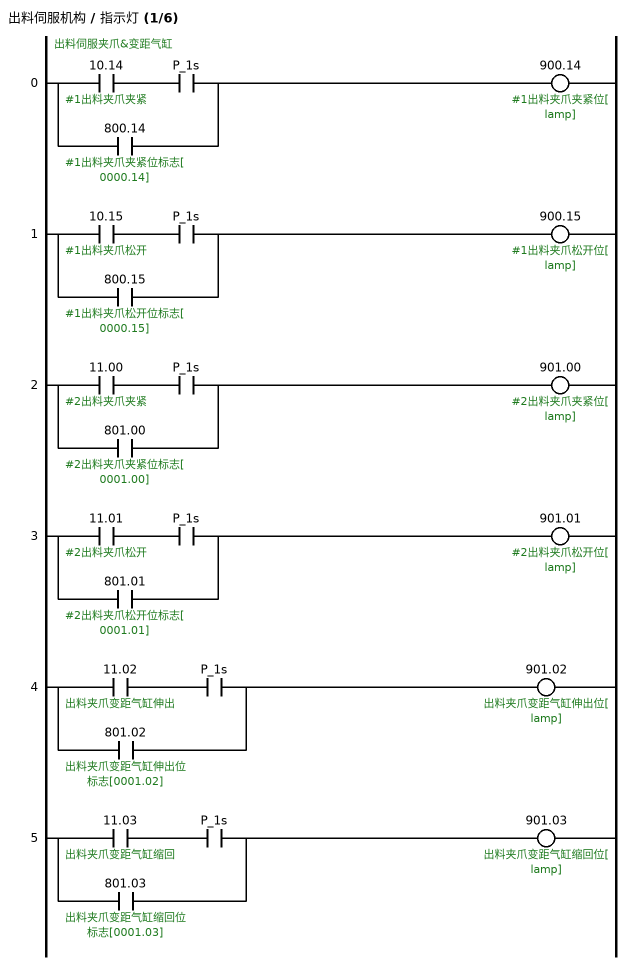
; [picture p504: 出料伺服机构 / 指示灯, rungs 0-5]
; rung 0: 出料伺服夹爪&变距气缸
LD 10.14  ; #1出料夹爪夹紧
AND P_1s
OR 800.14  ; #1出料夹爪夹紧位标志[0000.14]
OUT 900.14  ; #1出料夹爪夹紧位[lamp]
; rung 1
LD 10.15  ; #1出料夹爪松开
AND P_1s
OR 800.15  ; #1出料夹爪松开位标志[0000.15]
OUT 900.15  ; #1出料夹爪松开位[lamp]
; rung 2
LD 11.00  ; #2出料夹爪夹紧
AND P_1s
OR 801.00  ; #2出料夹爪夹紧位标志[0001.00]
OUT 901.00  ; #2出料夹爪夹紧位[lamp]
; rung 3
LD 11.01  ; #2出料夹爪松开
AND P_1s
OR 801.01  ; #2出料夹爪松开位标志[0001.01]
OUT 901.01  ; #2出料夹爪松开位[lamp]
; rung 4
LD 11.02  ; 出料夹爪变距气缸伸出
AND P_1s
OR 801.02  ; 出料夹爪变距气缸伸出位标志[0001.02]
OUT 901.02  ; 出料夹爪变距气缸伸出位[lamp]
; rung 5
LD 11.03  ; 出料夹爪变距气缸缩回
AND P_1s
OR 801.03  ; 出料夹爪变距气缸缩回位标志[0001.03]
OUT 901.03  ; 出料夹爪变距气缸缩回位[lamp]

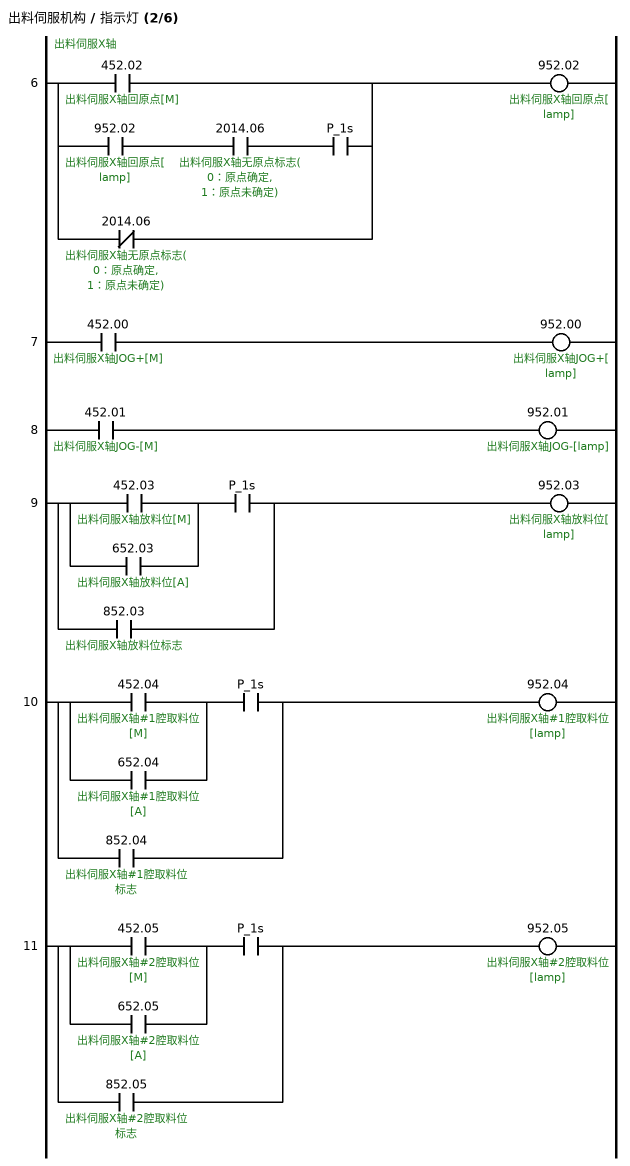
; rung 6: 出料伺服X轴
LD 452.02  ; 出料伺服X轴回原点[M]
LD 952.02  ; 出料伺服X轴回原点[lamp]
AND 2014.06  ; 出料伺服X轴无原点标志(0：原点确定,1：原点未确定)
AND P_1s
ORLD
ORNOT 2014.06  ; 出料伺服X轴无原点标志(0：原点确定,1：原点未确定)
OUT 952.02  ; 出料伺服X轴回原点[lamp]
; rung 7
LD 452.00  ; 出料伺服X轴JOG+[M]
OUT 952.00  ; 出料伺服X轴JOG+[lamp]
; rung 8
LD 452.01  ; 出料伺服X轴JOG-[M]
OUT 952.01  ; 出料伺服X轴JOG-[lamp]
; rung 9
LD 452.03  ; 出料伺服X轴放料位[M]
OR 652.03  ; 出料伺服X轴放料位[A]
AND P_1s
OR 852.03  ; 出料伺服X轴放料位标志
OUT 952.03  ; 出料伺服X轴放料位[lamp]
; rung 10
LD 452.04  ; 出料伺服X轴#1腔取料位[M]
OR 652.04  ; 出料伺服X轴#1腔取料位[A]
AND P_1s
OR 852.04  ; 出料伺服X轴#1腔取料位标志
OUT 952.04  ; 出料伺服X轴#1腔取料位[lamp]
; rung 11
LD 452.05  ; 出料伺服X轴#2腔取料位[M]
OR 652.05  ; 出料伺服X轴#2腔取料位[A]
AND P_1s
OR 852.05  ; 出料伺服X轴#2腔取料位标志
OUT 952.05  ; 出料伺服X轴#2腔取料位[lamp]

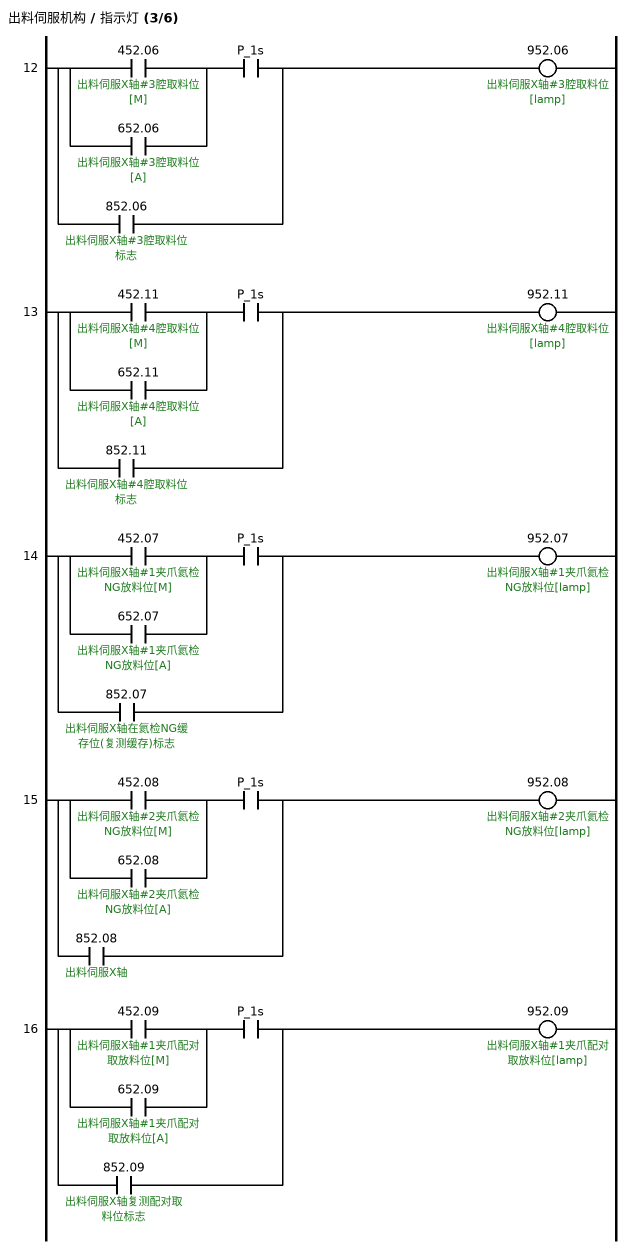
; rung 12
LD 452.06  ; 出料伺服X轴#3腔取料位[M]
OR 652.06  ; 出料伺服X轴#3腔取料位[A]
AND P_1s
OR 852.06  ; 出料伺服X轴#3腔取料位标志
OUT 952.06  ; 出料伺服X轴#3腔取料位[lamp]
; rung 13
LD 452.11  ; 出料伺服X轴#4腔取料位[M]
OR 652.11  ; 出料伺服X轴#4腔取料位[A]
AND P_1s
OR 852.11  ; 出料伺服X轴#4腔取料位标志
OUT 952.11  ; 出料伺服X轴#4腔取料位[lamp]
; rung 14
LD 452.07  ; 出料伺服X轴#1夹爪氦检NG放料位[M]
OR 652.07  ; 出料伺服X轴#1夹爪氦检NG放料位[A]
AND P_1s
OR 852.07  ; 出料伺服X轴在氦检NG缓存位(复测缓存)标志
OUT 952.07  ; 出料伺服X轴#1夹爪氦检NG放料位[lamp]
; rung 15
LD 452.08  ; 出料伺服X轴#2夹爪氦检NG放料位[M]
OR 652.08  ; 出料伺服X轴#2夹爪氦检NG放料位[A]
AND P_1s
OR 852.08  ; 出料伺服X轴
OUT 952.08  ; 出料伺服X轴#2夹爪氦检NG放料位[lamp]
; rung 16
LD 452.09  ; 出料伺服X轴#1夹爪配对取放料位[M]
OR 652.09  ; 出料伺服X轴#1夹爪配对取放料位[A]
AND P_1s
OR 852.09  ; 出料伺服X轴复测配对取料位标志
OUT 952.09  ; 出料伺服X轴#1夹爪配对取放料位[lamp]

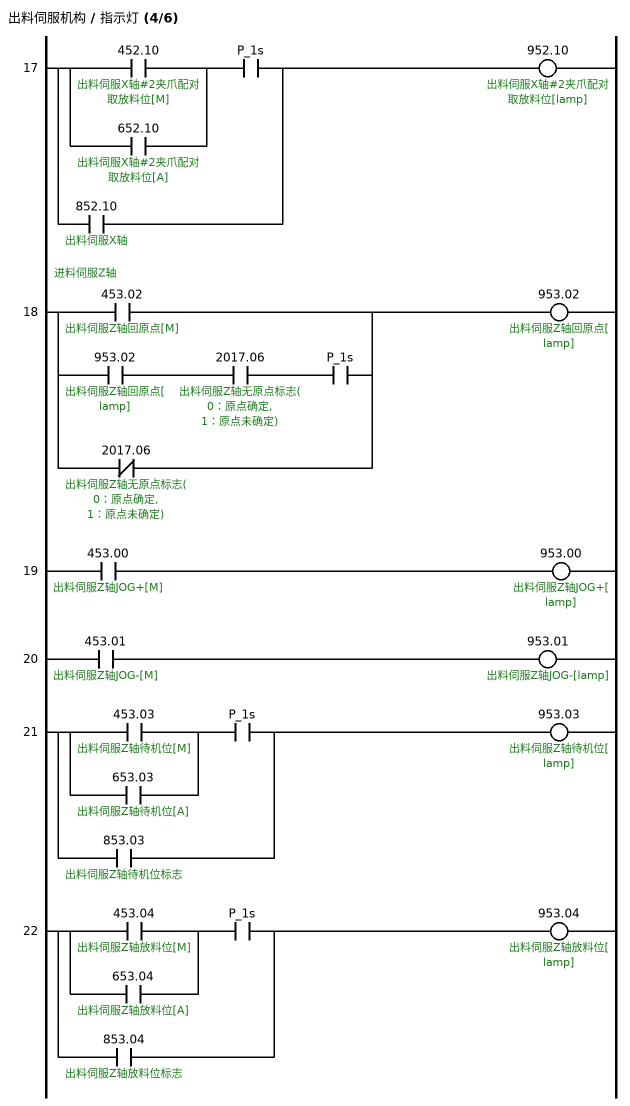
; rung 17
LD 452.10  ; 出料伺服X轴#2夹爪配对取放料位[M]
OR 652.10  ; 出料伺服X轴#2夹爪配对取放料位[A]
AND P_1s
OR 852.10  ; 出料伺服X轴
OUT 952.10  ; 出料伺服X轴#2夹爪配对取放料位[lamp]
; rung 18: 进料伺服Z轴
LD 453.02  ; 出料伺服Z轴回原点[M]
LD 953.02  ; 出料伺服Z轴回原点[lamp]
AND 2017.06  ; 出料伺服Z轴无原点标志(0：原点确定,1：原点未确定)
AND P_1s
ORLD
ORNOT 2017.06  ; 出料伺服Z轴无原点标志(0：原点确定,1：原点未确定)
OUT 953.02  ; 出料伺服Z轴回原点[lamp]
; rung 19
LD 453.00  ; 出料伺服Z轴JOG+[M]
OUT 953.00  ; 出料伺服Z轴JOG+[lamp]
; rung 20
LD 453.01  ; 出料伺服Z轴JOG-[M]
OUT 953.01  ; 出料伺服Z轴JOG-[lamp]
; rung 21
LD 453.03  ; 出料伺服Z轴待机位[M]
OR 653.03  ; 出料伺服Z轴待机位[A]
AND P_1s
OR 853.03  ; 出料伺服Z轴待机位标志
OUT 953.03  ; 出料伺服Z轴待机位[lamp]
; rung 22
LD 453.04  ; 出料伺服Z轴放料位[M]
OR 653.04  ; 出料伺服Z轴放料位[A]
AND P_1s
OR 853.04  ; 出料伺服Z轴放料位标志
OUT 953.04  ; 出料伺服Z轴放料位[lamp]

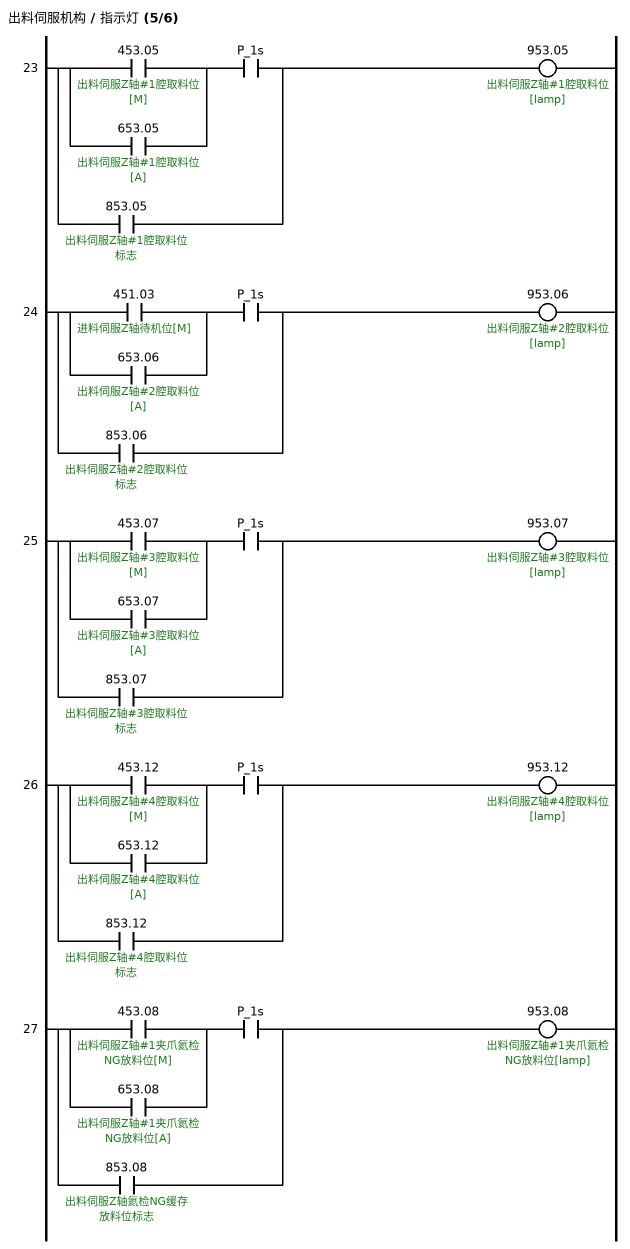
; rung 23
LD 453.05  ; 出料伺服Z轴#1腔取料位[M]
OR 653.05  ; 出料伺服Z轴#1腔取料位[A]
AND P_1s
OR 853.05  ; 出料伺服Z轴#1腔取料位标志
OUT 953.05  ; 出料伺服Z轴#1腔取料位[lamp]
; rung 24
LD 451.03  ; 进料伺服Z轴待机位[M]
OR 653.06  ; 出料伺服Z轴#2腔取料位[A]
AND P_1s
OR 853.06  ; 出料伺服Z轴#2腔取料位标志
OUT 953.06  ; 出料伺服Z轴#2腔取料位[lamp]
; rung 25
LD 453.07  ; 出料伺服Z轴#3腔取料位[M]
OR 653.07  ; 出料伺服Z轴#3腔取料位[A]
AND P_1s
OR 853.07  ; 出料伺服Z轴#3腔取料位标志
OUT 953.07  ; 出料伺服Z轴#3腔取料位[lamp]
; rung 26
LD 453.12  ; 出料伺服Z轴#4腔取料位[M]
OR 653.12  ; 出料伺服Z轴#4腔取料位[A]
AND P_1s
OR 853.12  ; 出料伺服Z轴#4腔取料位标志
OUT 953.12  ; 出料伺服Z轴#4腔取料位[lamp]
; rung 27
LD 453.08  ; 出料伺服Z轴#1夹爪氦检NG放料位[M]
OR 653.08  ; 出料伺服Z轴#1夹爪氦检NG放料位[A]
AND P_1s
OR 853.08  ; 出料伺服Z轴氦检NG缓存放料位标志
OUT 953.08  ; 出料伺服Z轴#1夹爪氦检NG放料位[lamp]

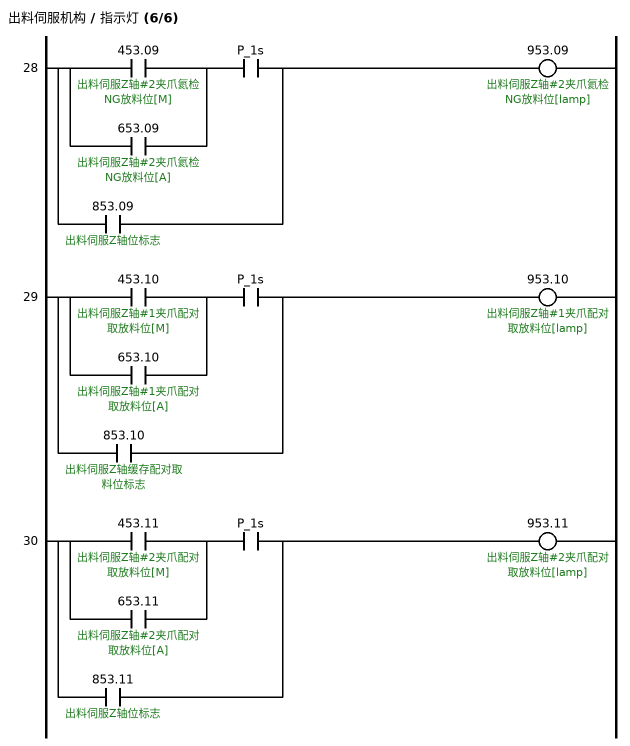
; rung 28
LD 453.09  ; 出料伺服Z轴#2夹爪氦检NG放料位[M]
OR 653.09  ; 出料伺服Z轴#2夹爪氦检NG放料位[A]
AND P_1s
OR 853.09  ; 出料伺服Z轴位标志
OUT 953.09  ; 出料伺服Z轴#2夹爪氦检NG放料位[lamp]
; rung 29
LD 453.10  ; 出料伺服Z轴#1夹爪配对取放料位[M]
OR 653.10  ; 出料伺服Z轴#1夹爪配对取放料位[A]
AND P_1s
OR 853.10  ; 出料伺服Z轴缓存配对取料位标志
OUT 953.10  ; 出料伺服Z轴#1夹爪配对取放料位[lamp]
; rung 30
LD 453.11  ; 出料伺服Z轴#2夹爪配对取放料位[M]
OR 653.11  ; 出料伺服Z轴#2夹爪配对取放料位[A]
AND P_1s
OR 853.11  ; 出料伺服Z轴位标志
OUT 953.11  ; 出料伺服Z轴#2夹爪配对取放料位[lamp]

### Section 外部输出

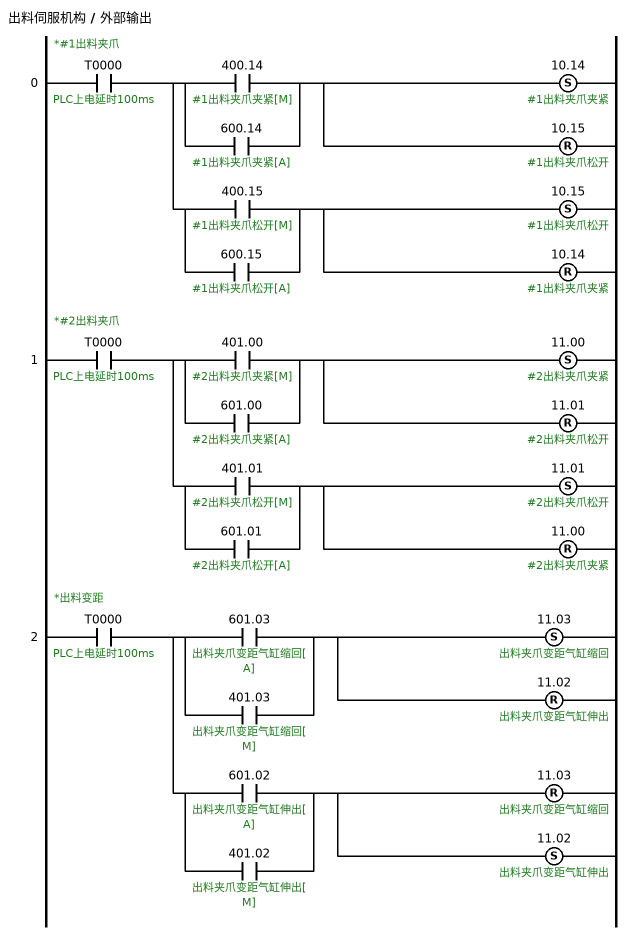
; rung 0: *#1出料夹爪
LD T0000  ; PLC上电延时100ms
OUT TR0
LD 400.14  ; #1出料夹爪夹紧[M]
OR 600.14  ; #1出料夹爪夹紧[A]
ANDLD
SET 10.14  ; #1出料夹爪夹紧
RSET 10.15  ; #1出料夹爪松开
LD TR0
LD 400.15  ; #1出料夹爪松开[M]
OR 600.15  ; #1出料夹爪松开[A]
ANDLD
SET 10.15  ; #1出料夹爪松开
RSET 10.14  ; #1出料夹爪夹紧
; rung 1: *#2出料夹爪
LD T0000  ; PLC上电延时100ms
OUT TR0
LD 401.00  ; #2出料夹爪夹紧[M]
OR 601.00  ; #2出料夹爪夹紧[A]
ANDLD
SET 11.00  ; #2出料夹爪夹紧
RSET 11.01  ; #2出料夹爪松开
LD TR0
LD 401.01  ; #2出料夹爪松开[M]
OR 601.01  ; #2出料夹爪松开[A]
ANDLD
SET 11.01  ; #2出料夹爪松开
RSET 11.00  ; #2出料夹爪夹紧
; rung 2: *出料变距
LD T0000  ; PLC上电延时100ms
OUT TR0
LD 601.03  ; 出料夹爪变距气缸缩回[A]
OR 401.03  ; 出料夹爪变距气缸缩回[M]
ANDLD
SET 11.03  ; 出料夹爪变距气缸缩回
RSET 11.02  ; 出料夹爪变距气缸伸出
LD TR0
LD 601.02  ; 出料夹爪变距气缸伸出[A]
OR 401.02  ; 出料夹爪变距气缸伸出[M]
ANDLD
RSET 11.03  ; 出料夹爪变距气缸缩回
SET 11.02  ; 出料夹爪变距气缸伸出

### Section END
; rung 0
END(001)

## Program NG缓存机构 (cyclic task 5)

### Section NG缓存

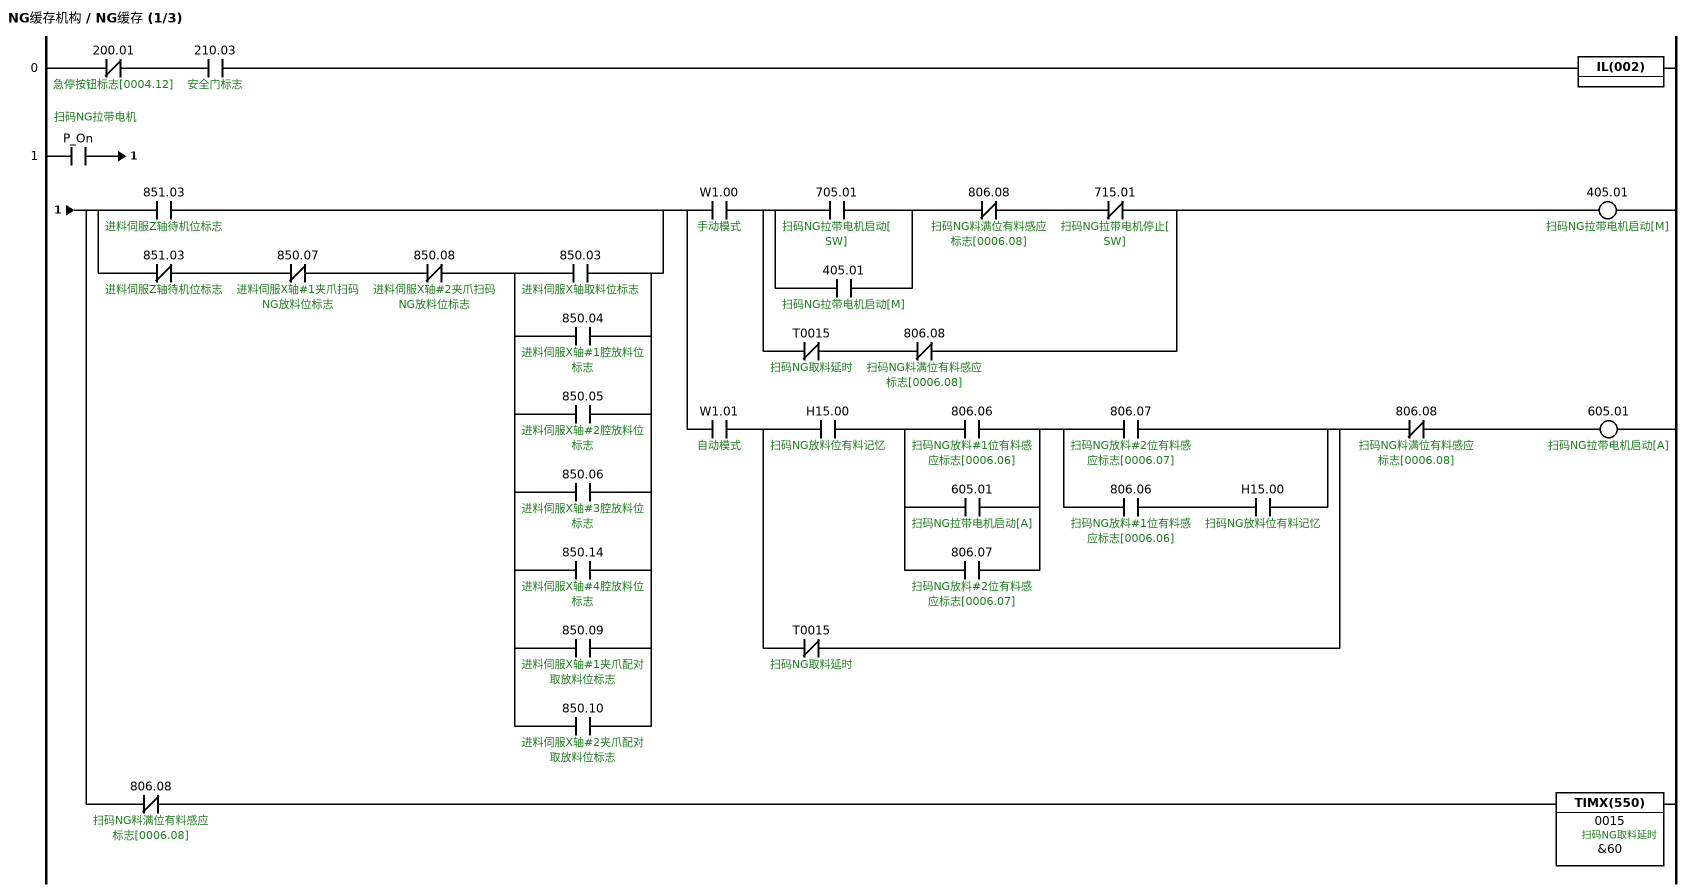
; rung 0
LDNOT 200.01  ; 急停按钮标志[0004.12]
AND 210.03  ; 安全门标志
IL(002)
; rung 1: 扫码NG拉带电机
LD P_On
OUT TR0
LD 851.03  ; 进料伺服Z轴待机位标志
LDNOT 851.03  ; 进料伺服Z轴待机位标志
ANDNOT 850.07  ; 进料伺服X轴#1夹爪扫码NG放料位标志
ANDNOT 850.08  ; 进料伺服X轴#2夹爪扫码NG放料位标志
LD 850.03  ; 进料伺服X轴取料位标志
OR 850.04  ; 进料伺服X轴#1腔放料位标志
OR 850.05  ; 进料伺服X轴#2腔放料位标志
OR 850.06  ; 进料伺服X轴#3腔放料位标志
OR 850.14  ; 进料伺服X轴#4腔放料位标志
OR 850.09  ; 进料伺服X轴#1夹爪配对取放料位标志
OR 850.10  ; 进料伺服X轴#2夹爪配对取放料位标志
ANDLD
ORLD
ANDLD
OUT TR1
AND W1.00  ; 手动模式
LD 705.01  ; 扫码NG拉带电机启动[SW]
OR 405.01  ; 扫码NG拉带电机启动[M]
ANDNOT 806.08  ; 扫码NG料满位有料感应标志[0006.08]
ANDNOT 715.01  ; 扫码NG拉带电机停止[SW]
LDNOT T0015  ; 扫码NG取料延时
ANDNOT 806.08  ; 扫码NG料满位有料感应标志[0006.08]
ORLD
ANDLD
OUT 405.01  ; 扫码NG拉带电机启动[M]
LD TR1
AND W1.01  ; 自动模式
LD H15.00  ; 扫码NG放料位有料记忆
LD 806.06  ; 扫码NG放料#1位有料感应标志[0006.06]
OR 605.01  ; 扫码NG拉带电机启动[A]
OR 806.07  ; 扫码NG放料#2位有料感应标志[0006.07]
ANDLD
LD 806.07  ; 扫码NG放料#2位有料感应标志[0006.07]
LD 806.06  ; 扫码NG放料#1位有料感应标志[0006.06]
AND H15.00  ; 扫码NG放料位有料记忆
ORLD
ANDLD
ORNOT T0015  ; 扫码NG取料延时
ANDLD
ANDNOT 806.08  ; 扫码NG料满位有料感应标志[0006.08]
OUT 605.01  ; 扫码NG拉带电机启动[A]
LD TR0
ANDNOT 806.08  ; 扫码NG料满位有料感应标志[0006.08]
TIMX(550) 0015 &60  ; 扫码NG取料延时

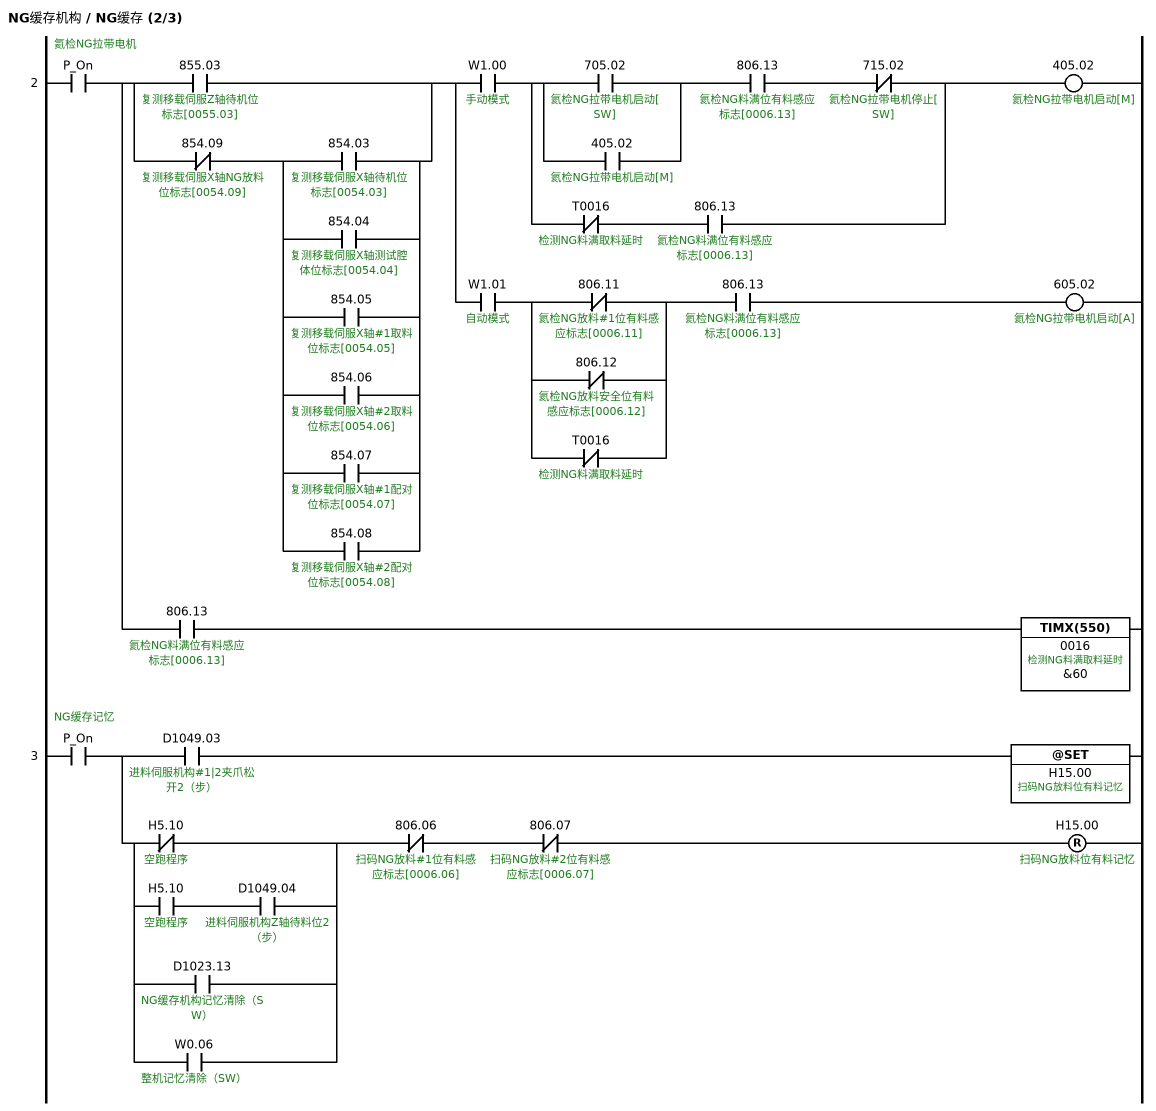
; rung 2: 氦检NG拉带电机
LD P_On
OUT TR0
LD 855.03  ; 复测移载伺服Z轴待机位标志[0055.03]
LDNOT 854.09  ; 复测移载伺服X轴NG放料位标志[0054.09]
LD 854.03  ; 复测移载伺服X轴待机位标志[0054.03]
OR 854.04  ; 复测移载伺服X轴测试腔体位标志[0054.04]
OR 854.05  ; 复测移载伺服X轴#1取料位标志[0054.05]
OR 854.06  ; 复测移载伺服X轴#2取料位标志[0054.06]
OR 854.07  ; 复测移载伺服X轴#1配对位标志[0054.07]
OR 854.08  ; 复测移载伺服X轴#2配对位标志[0054.08]
ANDLD
ORLD
ANDLD
OUT TR1
AND W1.00  ; 手动模式
LD 705.02  ; 氦检NG拉带电机启动[SW]
OR 405.02  ; 氦检NG拉带电机启动[M]
AND 806.13  ; 氦检NG料满位有料感应标志[0006.13]
ANDNOT 715.02  ; 氦检NG拉带电机停止[SW]
LDNOT T0016  ; 检测NG料满取料延时
AND 806.13  ; 氦检NG料满位有料感应标志[0006.13]
ORLD
ANDLD
OUT 405.02  ; 氦检NG拉带电机启动[M]
LD TR1
AND W1.01  ; 自动模式
LDNOT 806.11  ; 氦检NG放料#1位有料感应标志[0006.11]
ORNOT 806.12  ; 氦检NG放料安全位有料感应标志[0006.12]
ORNOT T0016  ; 检测NG料满取料延时
ANDLD
AND 806.13  ; 氦检NG料满位有料感应标志[0006.13]
OUT 605.02  ; 氦检NG拉带电机启动[A]
LD TR0
AND 806.13  ; 氦检NG料满位有料感应标志[0006.13]
TIMX(550) 0016 &60  ; 检测NG料满取料延时
; rung 3: NG缓存记忆
LD P_On
OUT TR0
AND D1049.03  ; 进料伺服机构#1|2夹爪松开2（步）
@SET H15.00  ; 扫码NG放料位有料记忆
LD TR0
LDNOT H5.10  ; 空跑程序
LD H5.10  ; 空跑程序
AND D1049.04  ; 进料伺服机构Z轴待料位2（步）
ORLD
OR D1023.13  ; NG缓存机构记忆清除（SW）
OR W0.06  ; 整机记忆清除（SW）
ANDLD
ANDNOT 806.06  ; 扫码NG放料#1位有料感应标志[0006.06]
ANDNOT 806.07  ; 扫码NG放料#2位有料感应标志[0006.07]
RSET H15.00  ; 扫码NG放料位有料记忆

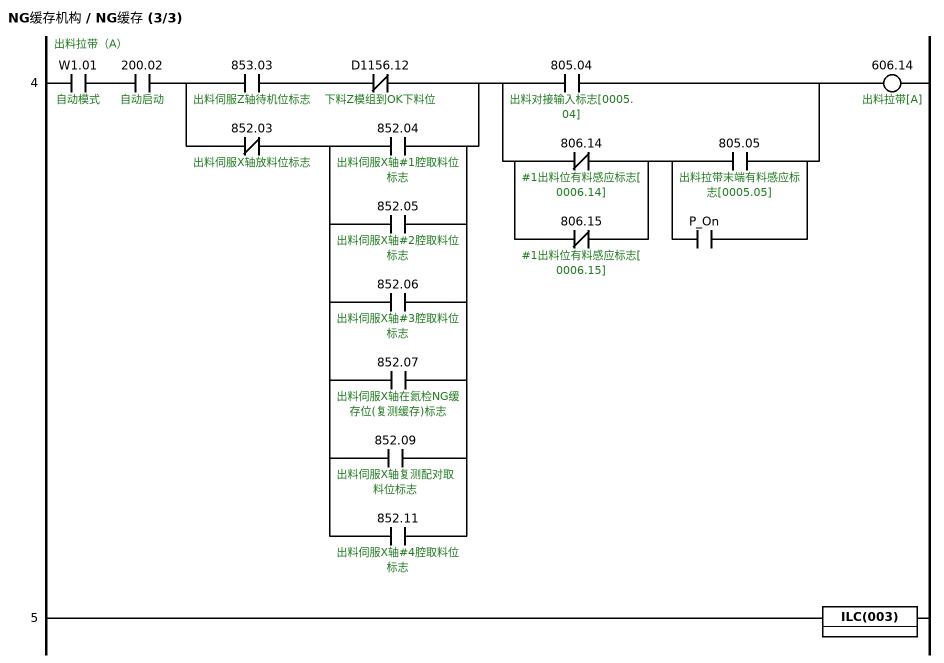
; rung 4: 出料拉带（A）
LD W1.01  ; 自动模式
AND 200.02  ; 自动启动
LD 853.03  ; 出料伺服Z轴待机位标志
ANDNOT D1156.12  ; 下料Z模组到OK下料位  // 拉带放料停止
LDNOT 852.03  ; 出料伺服X轴放料位标志
LD 852.04  ; 出料伺服X轴#1腔取料位标志
OR 852.05  ; 出料伺服X轴#2腔取料位标志
OR 852.06  ; 出料伺服X轴#3腔取料位标志
OR 852.07  ; 出料伺服X轴在氦检NG缓存位(复测缓存)标志
OR 852.09  ; 出料伺服X轴复测配对取料位标志
OR 852.11  ; 出料伺服X轴#4腔取料位标志
ANDLD
ORLD
ANDLD
LD 805.04  ; 出料对接输入标志[0005.04]
LDNOT 806.14  ; #1出料位有料感应标志[0006.14]
ORNOT 806.15  ; #1出料位有料感应标志[0006.15]
LD 805.05  ; 出料拉带末端有料感应标志[0005.05]  // 待确定是否需要增加感应器进行隔离，防止出现跟料现象（20190513）
OR P_On
ANDLD
ORLD
ANDLD
OUT 606.14  ; 出料拉带[A]
; rung 5
ILC(003)

### Section 外部输出

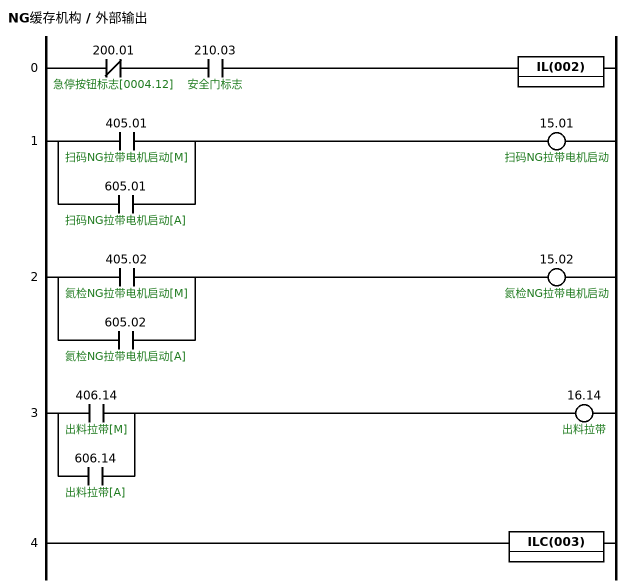
; rung 0
LDNOT 200.01  ; 急停按钮标志[0004.12]
AND 210.03  ; 安全门标志
IL(002)
; rung 1
LD 405.01  ; 扫码NG拉带电机启动[M]
OR 605.01  ; 扫码NG拉带电机启动[A]
OUT 15.01  ; 扫码NG拉带电机启动
; rung 2
LD 405.02  ; 氦检NG拉带电机启动[M]
OR 605.02  ; 氦检NG拉带电机启动[A]
OUT 15.02  ; 氦检NG拉带电机启动
; rung 3
LD 406.14  ; 出料拉带[M]
OR 606.14  ; 出料拉带[A]
OUT 16.14  ; 出料拉带
; rung 4
ILC(003)

### Section END
; rung 0
END(001)

## Program 复测移载机构 (cyclic task 6)

### Section Main

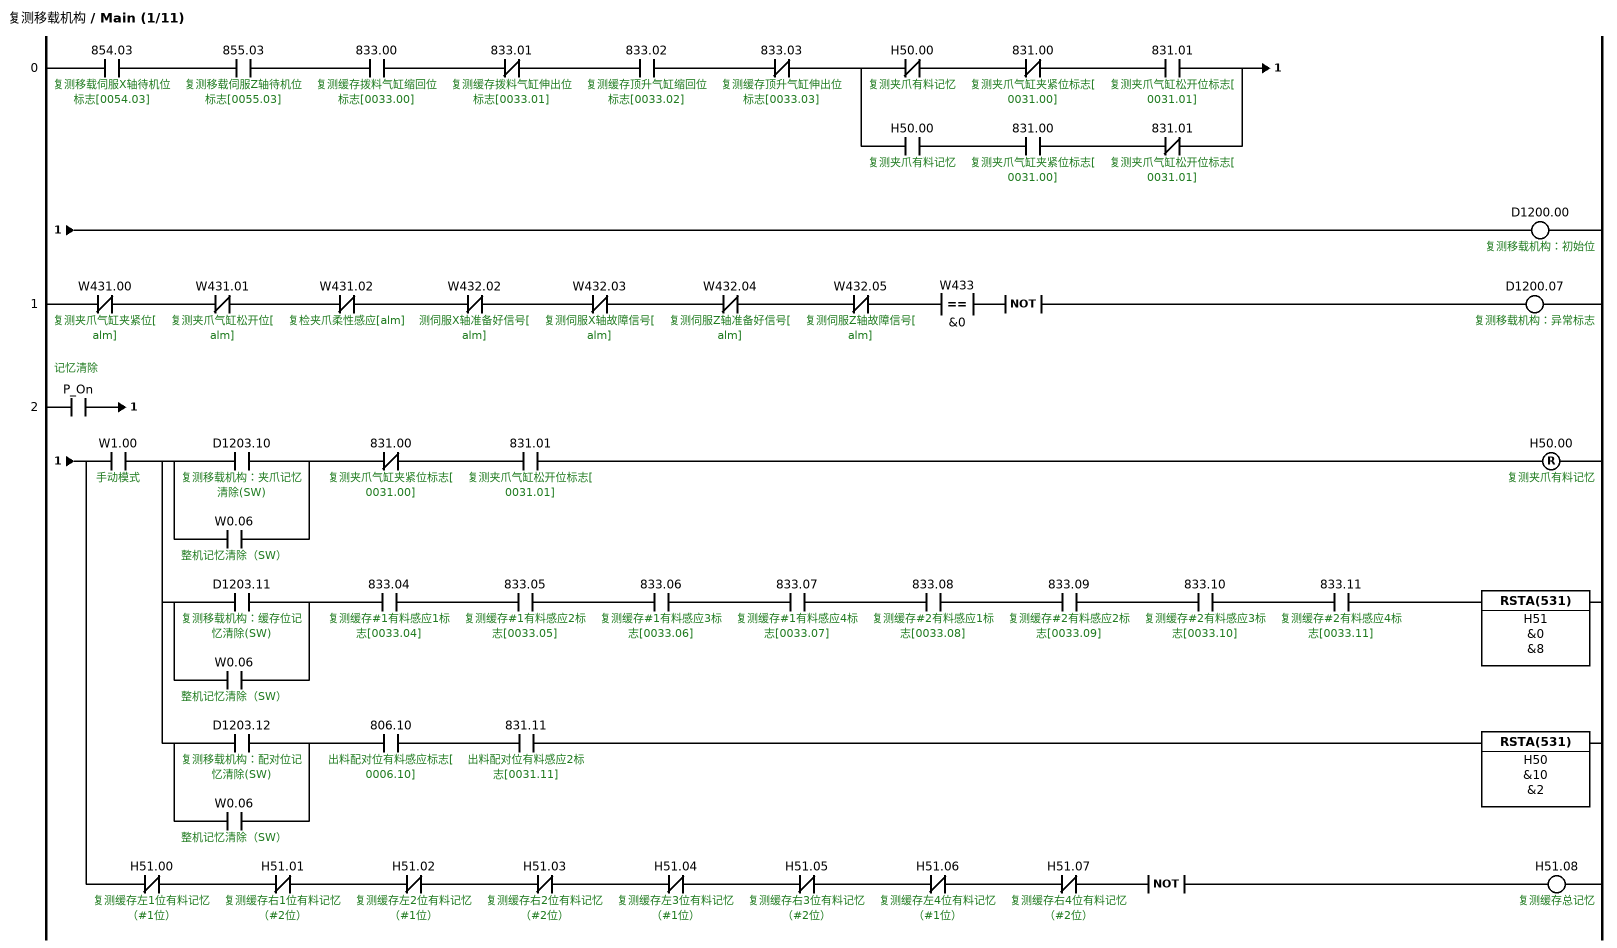
; rung 0
LD 854.03  ; 复测移载伺服X轴待机位标志[0054.03]
AND 855.03  ; 复测移载伺服Z轴待机位标志[0055.03]
AND 833.00  ; 复测缓存拨料气缸缩回位标志[0033.00]
ANDNOT 833.01  ; 复测缓存拨料气缸伸出位标志[0033.01]
AND 833.02  ; 复测缓存顶升气缸缩回位标志[0033.02]
ANDNOT 833.03  ; 复测缓存顶升气缸伸出位标志[0033.03]
LDNOT H50.00  ; 复测夹爪有料记忆
ANDNOT 831.00  ; 复测夹爪气缸夹紧位标志[0031.00]
AND 831.01  ; 复测夹爪气缸松开位标志[0031.01]
LD H50.00  ; 复测夹爪有料记忆
AND 831.00  ; 复测夹爪气缸夹紧位标志[0031.00]
ANDNOT 831.01  ; 复测夹爪气缸松开位标志[0031.01]
ORLD
ANDLD
OUT D1200.00  ; 复测移载机构：初始位
; rung 1
LDNOT W431.00  ; 复测夹爪气缸夹紧位[alm]
ANDNOT W431.01  ; 复测夹爪气缸松开位[alm]
ANDNOT W431.02  ; 复检夹爪柔性感应[alm]
ANDNOT W432.02  ; 测伺服X轴准备好信号[alm]
ANDNOT W432.03  ; 复测伺服X轴故障信号[alm]
ANDNOT W432.04  ; 复测伺服Z轴准备好信号[alm]
ANDNOT W432.05  ; 复测伺服Z轴故障信号[alm]
AND=(300) W433 &0
NOT(520)
OUT D1200.07  ; 复测移载机构：异常标志
; rung 2: 记忆清除
LD P_On
OUT TR0
AND W1.00  ; 手动模式
OUT TR1
LD D1203.10  ; 复测移载机构：夹爪记忆清除(SW)
OR W0.06  ; 整机记忆清除（SW）
ANDLD
ANDNOT 831.00  ; 复测夹爪气缸夹紧位标志[0031.00]
AND 831.01  ; 复测夹爪气缸松开位标志[0031.01]
RSET H50.00  ; 复测夹爪有料记忆
LD TR1
LD D1203.11  ; 复测移载机构：缓存位记忆清除(SW)
OR W0.06  ; 整机记忆清除（SW）
ANDLD
AND 833.04  ; 复测缓存#1有料感应1标志[0033.04]
AND 833.05  ; 复测缓存#1有料感应2标志[0033.05]
AND 833.06  ; 复测缓存#1有料感应3标志[0033.06]
AND 833.07  ; 复测缓存#1有料感应4标志[0033.07]
AND 833.08  ; 复测缓存#2有料感应1标志[0033.08]
AND 833.09  ; 复测缓存#2有料感应2标志[0033.09]
AND 833.10  ; 复测缓存#2有料感应3标志[0033.10]
AND 833.11  ; 复测缓存#2有料感应4标志[0033.11]
RSTA(531) H51 &0 &8
LD TR1
LD D1203.12  ; 复测移载机构：配对位记忆清除(SW)
OR W0.06  ; 整机记忆清除（SW）
ANDLD
AND 806.10  ; 出料配对位有料感应标志[0006.10]
AND 831.11  ; 出料配对位有料感应2标志[0031.11]
RSTA(531) H50 &10 &2
LD TR0
ANDNOT H51.00  ; 复测缓存左1位有料记忆（#1位）
ANDNOT H51.01  ; 复测缓存右1位有料记忆（#2位）
ANDNOT H51.02  ; 复测缓存左2位有料记忆（#1位）
ANDNOT H51.03  ; 复测缓存右2位有料记忆（#2位）
ANDNOT H51.04  ; 复测缓存左3位有料记忆（#1位）
ANDNOT H51.05  ; 复测缓存右3位有料记忆（#2位）
ANDNOT H51.06  ; 复测缓存左4位有料记忆（#1位）
ANDNOT H51.07  ; 复测缓存右4位有料记忆（#2位）
NOT(520)
OUT H51.08  ; 复测缓存总记忆

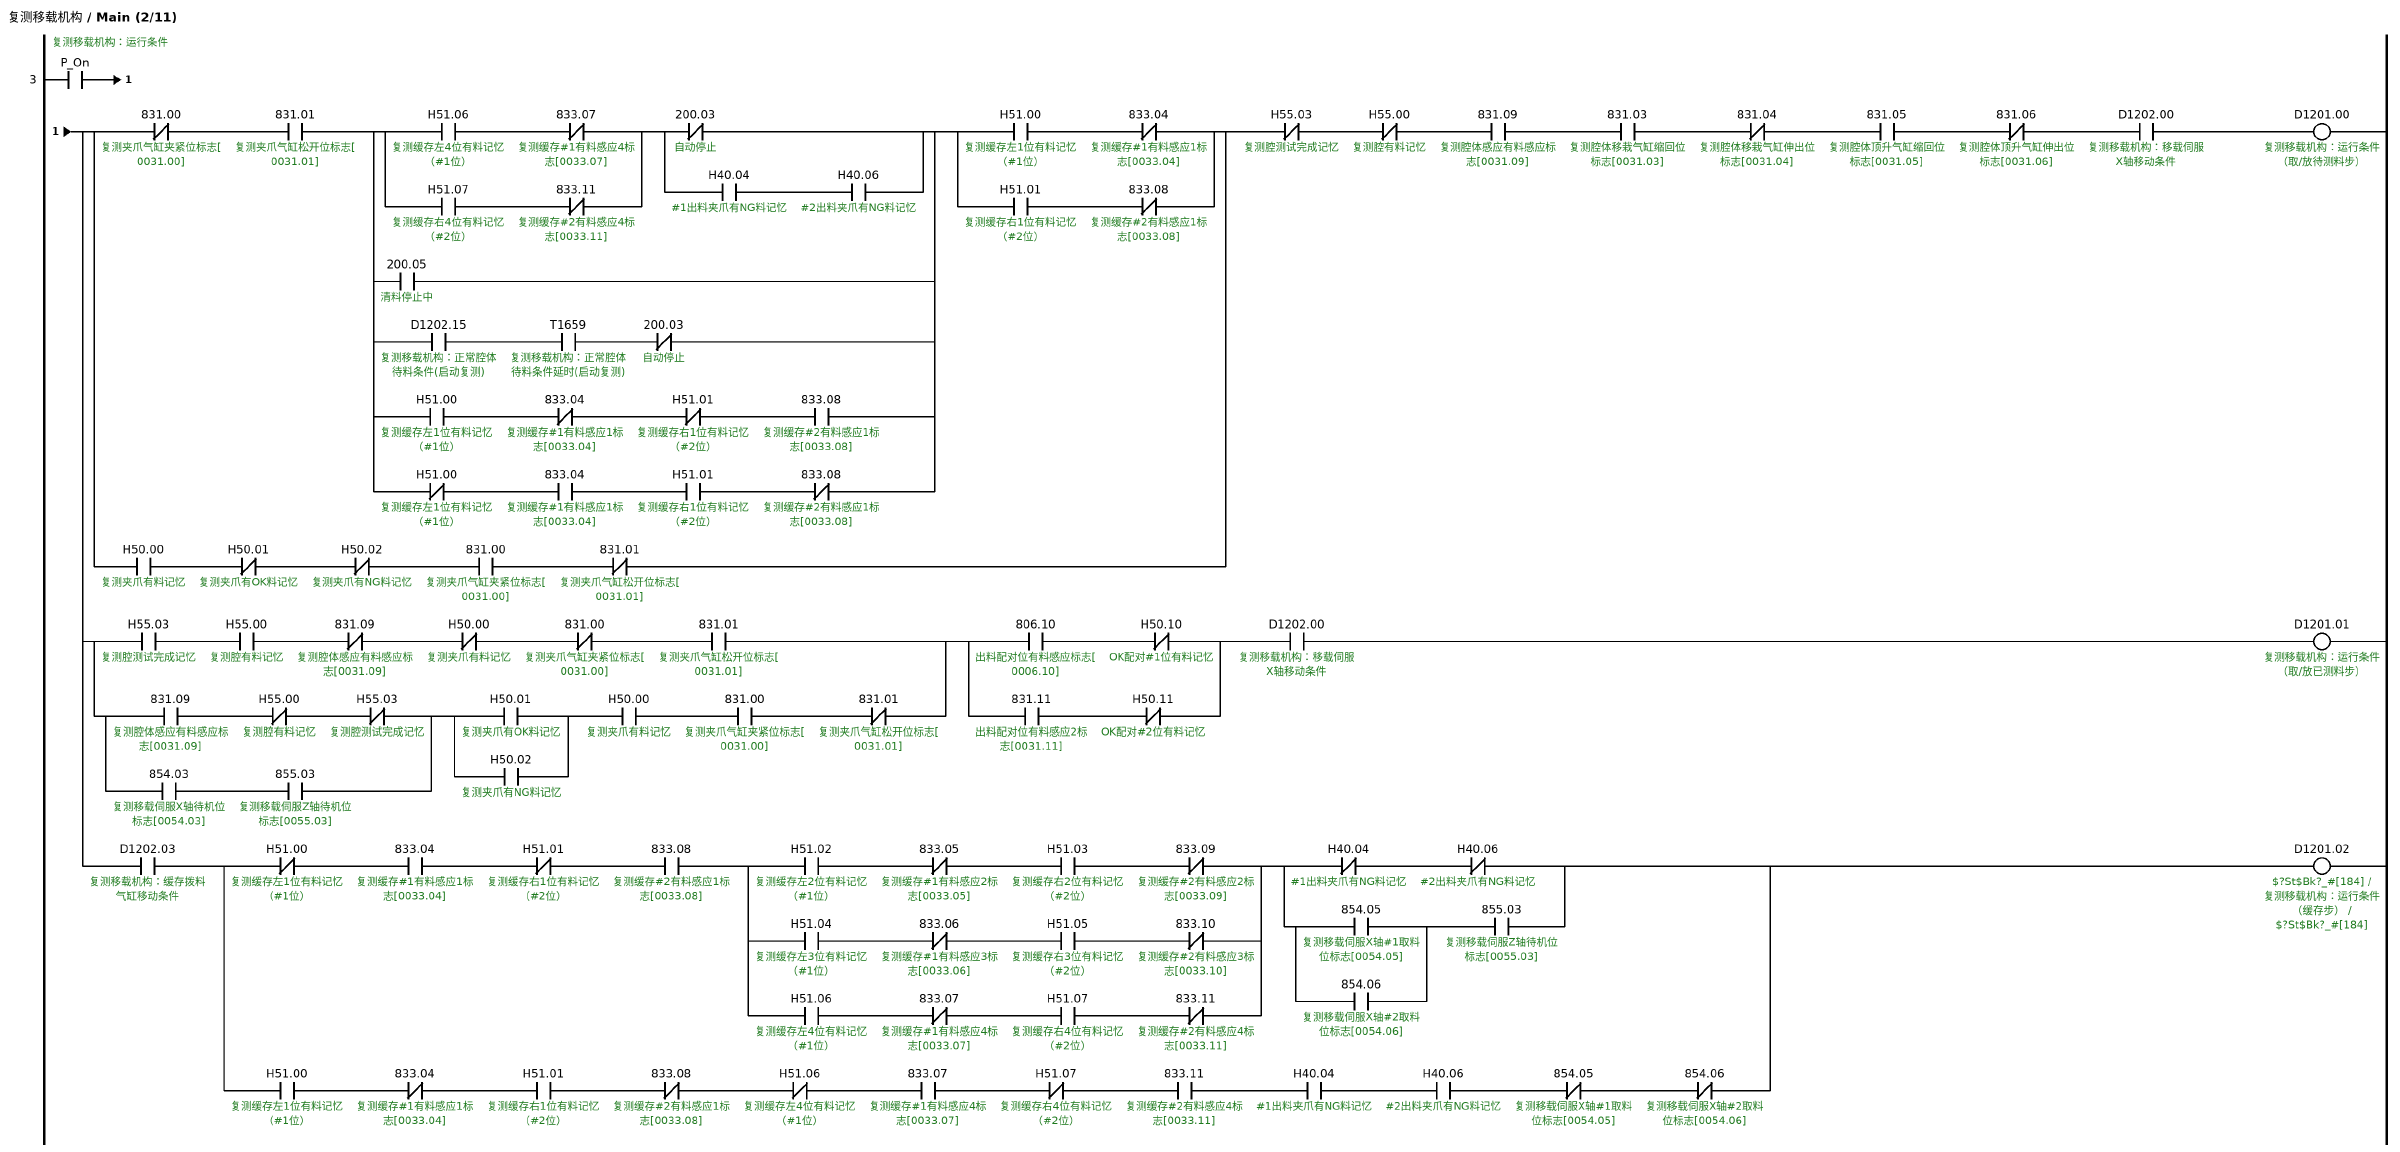
; rung 3: 复测移载机构：运行条件
LD P_On
OUT TR0
LDNOT 831.00  ; 复测夹爪气缸夹紧位标志[0031.00]
AND 831.01  ; 复测夹爪气缸松开位标志[0031.01]
LD H51.06  ; 复测缓存左4位有料记忆（#1位）  // 缓存料满则需提前进行复测
ANDNOT 833.07  ; 复测缓存#1有料感应4标志[0033.07]
LD H51.07  ; 复测缓存右4位有料记忆（#2位）
ANDNOT 833.11  ; 复测缓存#2有料感应4标志[0033.11]
ORLD
LDNOT 200.03  ; 自动停止
LD H40.04  ; #1出料夹爪有NG料记忆
AND H40.06  ; #2出料夹爪有NG料记忆
ORLD
ANDLD
OR 200.05  ; 清料停止中
LD D1202.15  ; 复测移载机构：正常腔体待料条件(启动复测)
AND T1659  ; 复测移载机构：正常腔体待料条件延时(启动复测)
ANDNOT 200.03  ; 自动停止
ORLD
LD H51.00  ; 复测缓存左1位有料记忆（#1位）  // 缓存第一位出现单料是需直接清掉，防止下次待测料无法进行单个放料
ANDNOT 833.04  ; 复测缓存#1有料感应1标志[0033.04]
ANDNOT H51.01  ; 复测缓存右1位有料记忆（#2位）
AND 833.08  ; 复测缓存#2有料感应1标志[0033.08]
ORLD
LDNOT H51.00  ; 复测缓存左1位有料记忆（#1位）
AND 833.04  ; 复测缓存#1有料感应1标志[0033.04]
AND H51.01  ; 复测缓存右1位有料记忆（#2位）
ANDNOT 833.08  ; 复测缓存#2有料感应1标志[0033.08]
ORLD
ANDLD
LD H51.00  ; 复测缓存左1位有料记忆（#1位）
ANDNOT 833.04  ; 复测缓存#1有料感应1标志[0033.04]
LD H51.01  ; 复测缓存右1位有料记忆（#2位）
ANDNOT 833.08  ; 复测缓存#2有料感应1标志[0033.08]
ORLD
ANDLD
LD H50.00  ; 复测夹爪有料记忆
ANDNOT H50.01  ; 复测夹爪有OK料记忆
ANDNOT H50.02  ; 复测夹爪有NG料记忆
AND 831.00  ; 复测夹爪气缸夹紧位标志[0031.00]
ANDNOT 831.01  ; 复测夹爪气缸松开位标志[0031.01]
ORLD
ANDLD
ANDNOT H55.03  ; 复测腔测试完成记忆
ANDNOT H55.00  ; 复测腔有料记忆
AND 831.09  ; 复测腔体感应有料感应标志[0031.09]
AND 831.03  ; 复测腔体移栽气缸缩回位标志[0031.03]
ANDNOT 831.04  ; 复测腔体移栽气缸伸出位标志[0031.04]
AND 831.05  ; 复测腔体顶升气缸缩回位标志[0031.05]
ANDNOT 831.06  ; 复测腔体顶升气缸伸出位标志[0031.06]
AND D1202.00  ; 复测移载机构：移载伺服X轴移动条件
OUT D1201.00  ; 复测移载机构：运行条件（取/放待测料步）
LD TR0
LD H55.03  ; 复测腔测试完成记忆
AND H55.00  ; 复测腔有料记忆
ANDNOT 831.09  ; 复测腔体感应有料感应标志[0031.09]
ANDNOT H50.00  ; 复测夹爪有料记忆
ANDNOT 831.00  ; 复测夹爪气缸夹紧位标志[0031.00]
AND 831.01  ; 复测夹爪气缸松开位标志[0031.01]
LD 831.09  ; 复测腔体感应有料感应标志[0031.09]
ANDNOT H55.00  ; 复测腔有料记忆
ANDNOT H55.03  ; 复测腔测试完成记忆
LD 854.03  ; 复测移载伺服X轴待机位标志[0054.03]
AND 855.03  ; 复测移载伺服Z轴待机位标志[0055.03]
ORLD
LD H50.01  ; 复测夹爪有OK料记忆
OR H50.02  ; 复测夹爪有NG料记忆
ANDLD
AND H50.00  ; 复测夹爪有料记忆
AND 831.00  ; 复测夹爪气缸夹紧位标志[0031.00]
ANDNOT 831.01  ; 复测夹爪气缸松开位标志[0031.01]
ORLD
ANDLD
LD 806.10  ; 出料配对位有料感应标志[0006.10]
ANDNOT H50.10  ; OK配对#1位有料记忆
LD 831.11  ; 出料配对位有料感应2标志[0031.11]
ANDNOT H50.11  ; OK配对#2位有料记忆
ORLD
ANDLD
AND D1202.00  ; 复测移载机构：移载伺服X轴移动条件
OUT D1201.01  ; 复测移载机构：运行条件（取/放已测料步）
LD TR0
AND D1202.03  ; 复测移载机构：缓存拨料气缸移动条件
LDNOT H51.00  ; 复测缓存左1位有料记忆（#1位）
AND 833.04  ; 复测缓存#1有料感应1标志[0033.04]
ANDNOT H51.01  ; 复测缓存右1位有料记忆（#2位）
AND 833.08  ; 复测缓存#2有料感应1标志[0033.08]
LD H51.02  ; 复测缓存左2位有料记忆（#1位）
ANDNOT 833.05  ; 复测缓存#1有料感应2标志[0033.05]
AND H51.03  ; 复测缓存右2位有料记忆（#2位）
ANDNOT 833.09  ; 复测缓存#2有料感应2标志[0033.09]
LD H51.04  ; 复测缓存左3位有料记忆（#1位）
ANDNOT 833.06  ; 复测缓存#1有料感应3标志[0033.06]
AND H51.05  ; 复测缓存右3位有料记忆（#2位）
ANDNOT 833.10  ; 复测缓存#2有料感应3标志[0033.10]
ORLD
LD H51.06  ; 复测缓存左4位有料记忆（#1位）
ANDNOT 833.07  ; 复测缓存#1有料感应4标志[0033.07]
AND H51.07  ; 复测缓存右4位有料记忆（#2位）
ANDNOT 833.11  ; 复测缓存#2有料感应4标志[0033.11]
ORLD
ANDLD
LDNOT H40.04  ; #1出料夹爪有NG料记忆
ANDNOT H40.06  ; #2出料夹爪有NG料记忆
LD 854.05  ; 复测移载伺服X轴#1取料位标志[0054.05]
OR 854.06  ; 复测移载伺服X轴#2取料位标志[0054.06]
AND 855.03  ; 复测移载伺服Z轴待机位标志[0055.03]
ORLD
ANDLD
LD H51.00  ; 复测缓存左1位有料记忆（#1位）
ANDNOT 833.04  ; 复测缓存#1有料感应1标志[0033.04]
AND H51.01  ; 复测缓存右1位有料记忆（#2位）
ANDNOT 833.08  ; 复测缓存#2有料感应1标志[0033.08]
ANDNOT H51.06  ; 复测缓存左4位有料记忆（#1位）
AND 833.07  ; 复测缓存#1有料感应4标志[0033.07]
ANDNOT H51.07  ; 复测缓存右4位有料记忆（#2位）
AND 833.11  ; 复测缓存#2有料感应4标志[0033.11]
AND H40.04  ; #1出料夹爪有NG料记忆
AND H40.06  ; #2出料夹爪有NG料记忆
ANDNOT 854.05  ; 复测移载伺服X轴#1取料位标志[0054.05]
ANDNOT 854.06  ; 复测移载伺服X轴#2取料位标志[0054.06]
ORLD
ANDLD
OUT D1201.02  ; $?St$Bk?_#[184] / 复测移载机构：运行条件（缓存步） / $?St$Bk?_#[184]

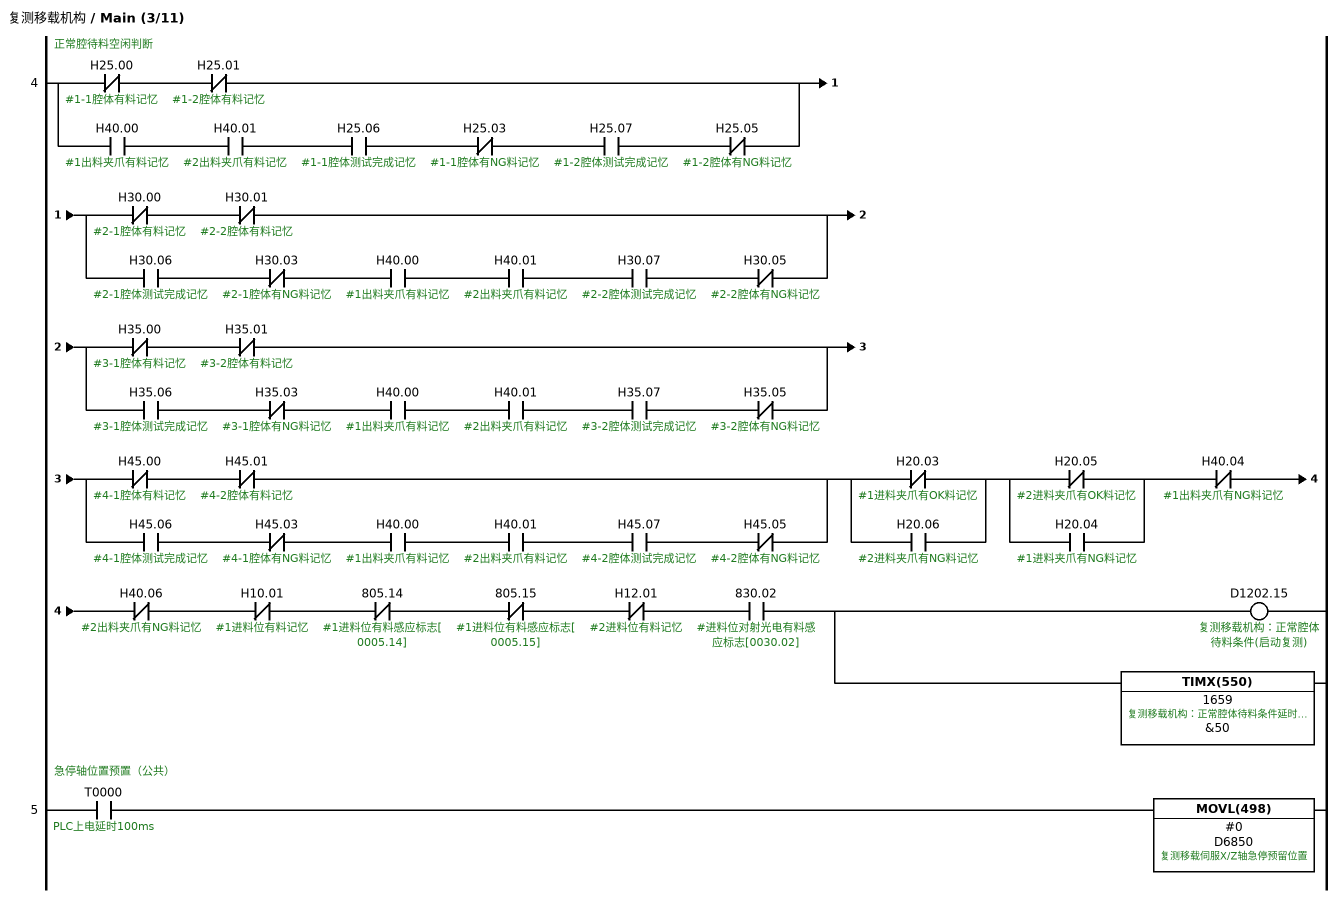
; rung 4: 正常腔待料空闲判断
LDNOT H25.00  ; #1-1腔体有料记忆
ANDNOT H25.01  ; #1-2腔体有料记忆
LD H40.00  ; #1出料夹爪有料记忆
AND H40.01  ; #2出料夹爪有料记忆
AND H25.06  ; #1-1腔体测试完成记忆
ANDNOT H25.03  ; #1-1腔体有NG料记忆
AND H25.07  ; #1-2腔体测试完成记忆
ANDNOT H25.05  ; #1-2腔体有NG料记忆
ORLD
LDNOT H30.00  ; #2-1腔体有料记忆
ANDNOT H30.01  ; #2-2腔体有料记忆
LD H30.06  ; #2-1腔体测试完成记忆
ANDNOT H30.03  ; #2-1腔体有NG料记忆
AND H40.00  ; #1出料夹爪有料记忆
AND H40.01  ; #2出料夹爪有料记忆
AND H30.07  ; #2-2腔体测试完成记忆
ANDNOT H30.05  ; #2-2腔体有NG料记忆
ORLD
ANDLD
LDNOT H35.00  ; #3-1腔体有料记忆
ANDNOT H35.01  ; #3-2腔体有料记忆
LD H35.06  ; #3-1腔体测试完成记忆
ANDNOT H35.03  ; #3-1腔体有NG料记忆
AND H40.00  ; #1出料夹爪有料记忆
AND H40.01  ; #2出料夹爪有料记忆
AND H35.07  ; #3-2腔体测试完成记忆
ANDNOT H35.05  ; #3-2腔体有NG料记忆
ORLD
ANDLD
LDNOT H45.00  ; #4-1腔体有料记忆
ANDNOT H45.01  ; #4-2腔体有料记忆
LD H45.06  ; #4-1腔体测试完成记忆
ANDNOT H45.03  ; #4-1腔体有NG料记忆
AND H40.00  ; #1出料夹爪有料记忆
AND H40.01  ; #2出料夹爪有料记忆
AND H45.07  ; #4-2腔体测试完成记忆
ANDNOT H45.05  ; #4-2腔体有NG料记忆
ORLD
ANDLD
LDNOT H20.03  ; #1进料夹爪有OK料记忆
OR H20.06  ; #2进料夹爪有NG料记忆
ANDLD
LDNOT H20.05  ; #2进料夹爪有OK料记忆
OR H20.04  ; #1进料夹爪有NG料记忆
ANDLD
ANDNOT H40.04  ; #1出料夹爪有NG料记忆
ANDNOT H40.06  ; #2出料夹爪有NG料记忆
ANDNOT H10.01  ; #1进料位有料记忆
ANDNOT 805.14  ; #1进料位有料感应标志[0005.14]
ANDNOT 805.15  ; #1进料位有料感应标志[0005.15]
ANDNOT H12.01  ; #2进料位有料记忆
AND 830.02  ; #进料位对射光电有料感应标志[0030.02]
OUT D1202.15  ; 复测移载机构：正常腔体待料条件(启动复测)
TIMX(550) 1659 &50  ; 复测移载机构：正常腔体待料条件延时(启动复测)
; rung 5: 急停轴位置预置（公共）
LD T0000  ; PLC上电延时100ms
MOVL(498) #0 D6850  ; 复测移载伺服X/Z轴急停预留位置

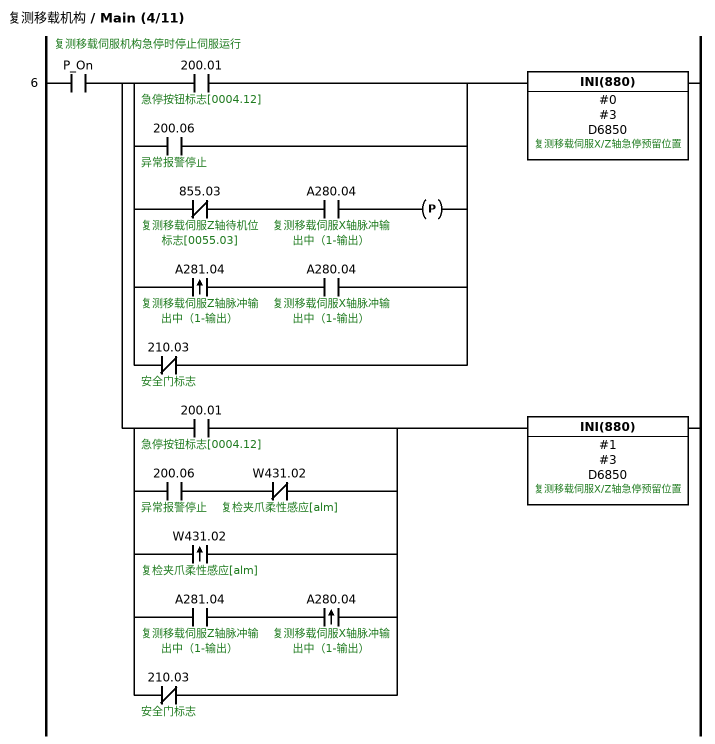
; rung 6: 复测移载伺服机构急停时停止伺服运行
LD P_On
OUT TR0
LD 200.01  ; 急停按钮标志[0004.12]
OR 200.06  ; 异常报警停止
LDNOT 855.03  ; 复测移载伺服Z轴待机位标志[0055.03]
AND A280.04  ; 复测移载伺服X轴脉冲输出中（1-输出）
UP(521)
ORLD
@LD A281.04  ; 复测移载伺服Z轴脉冲输出中（1-输出）
AND A280.04  ; 复测移载伺服X轴脉冲输出中（1-输出）
ORLD
ORNOT 210.03  ; 安全门标志
ANDLD
INI(880) #0 #3 D6850  ; 复测移载伺服X/Z轴急停预留位置  // 复测移载伺服X轴
LD TR0
LD 200.01  ; 急停按钮标志[0004.12]
LD 200.06  ; 异常报警停止
ANDNOT W431.02  ; 复检夹爪柔性感应[alm]
ORLD
@OR W431.02  ; 复检夹爪柔性感应[alm]
LD A281.04  ; 复测移载伺服Z轴脉冲输出中（1-输出）
@AND A280.04  ; 复测移载伺服X轴脉冲输出中（1-输出）
ORLD
ORNOT 210.03  ; 安全门标志
ANDLD
INI(880) #1 #3 D6850  ; 复测移载伺服X/Z轴急停预留位置  // 复测移载伺服Z轴

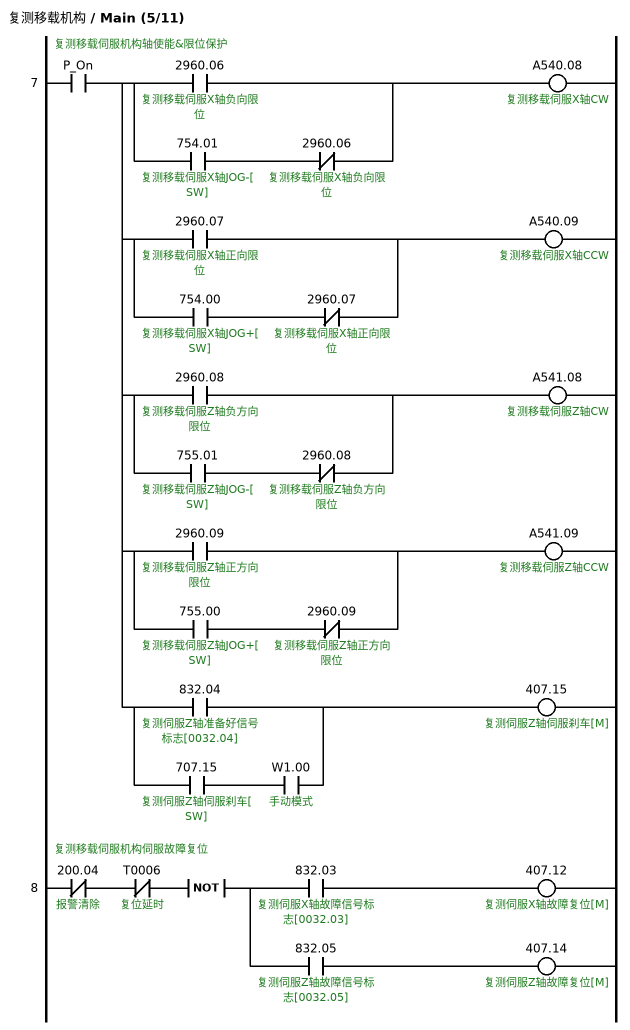
; rung 7: 复测移载伺服机构轴使能&限位保护
LD P_On
OUT TR0
LD 2960.06  ; 复测移载伺服X轴负向限位
LD 754.01  ; 复测移载伺服X轴JOG-[SW]
ANDNOT 2960.06  ; 复测移载伺服X轴负向限位
ORLD
ANDLD
OUT A540.08  ; 复测移载伺服X轴CW
LD TR0
LD 2960.07  ; 复测移载伺服X轴正向限位
LD 754.00  ; 复测移载伺服X轴JOG+[SW]
ANDNOT 2960.07  ; 复测移载伺服X轴正向限位
ORLD
ANDLD
OUT A540.09  ; 复测移载伺服X轴CCW
LD TR0
LD 2960.08  ; 复测移载伺服Z轴负方向限位
LD 755.01  ; 复测移载伺服Z轴JOG-[SW]
ANDNOT 2960.08  ; 复测移载伺服Z轴负方向限位
ORLD
ANDLD
OUT A541.08  ; 复测移载伺服Z轴CW
LD TR0
LD 2960.09  ; 复测移载伺服Z轴正方向限位
LD 755.00  ; 复测移载伺服Z轴JOG+[SW]
ANDNOT 2960.09  ; 复测移载伺服Z轴正方向限位
ORLD
ANDLD
OUT A541.09  ; 复测移载伺服Z轴CCW
LD TR0
LD 832.04  ; 复测伺服Z轴准备好信号标志[0032.04]
LD 707.15  ; 复测伺服Z轴伺服刹车[SW]
AND W1.00  ; 手动模式
ORLD
ANDLD
OUT 407.15  ; 复测伺服Z轴伺服刹车[M]
; rung 8: 复测移载伺服机构伺服故障复位
LDNOT 200.04  ; 报警清除
ANDNOT T0006  ; 复位延时
NOT(520)
OUT TR0
AND 832.03  ; 复测伺服X轴故障信号标志[0032.03]
OUT 407.12  ; 复测伺服X轴故障复位[M]
LD TR0
AND 832.05  ; 复测伺服Z轴故障信号标志[0032.05]
OUT 407.14  ; 复测伺服Z轴故障复位[M]

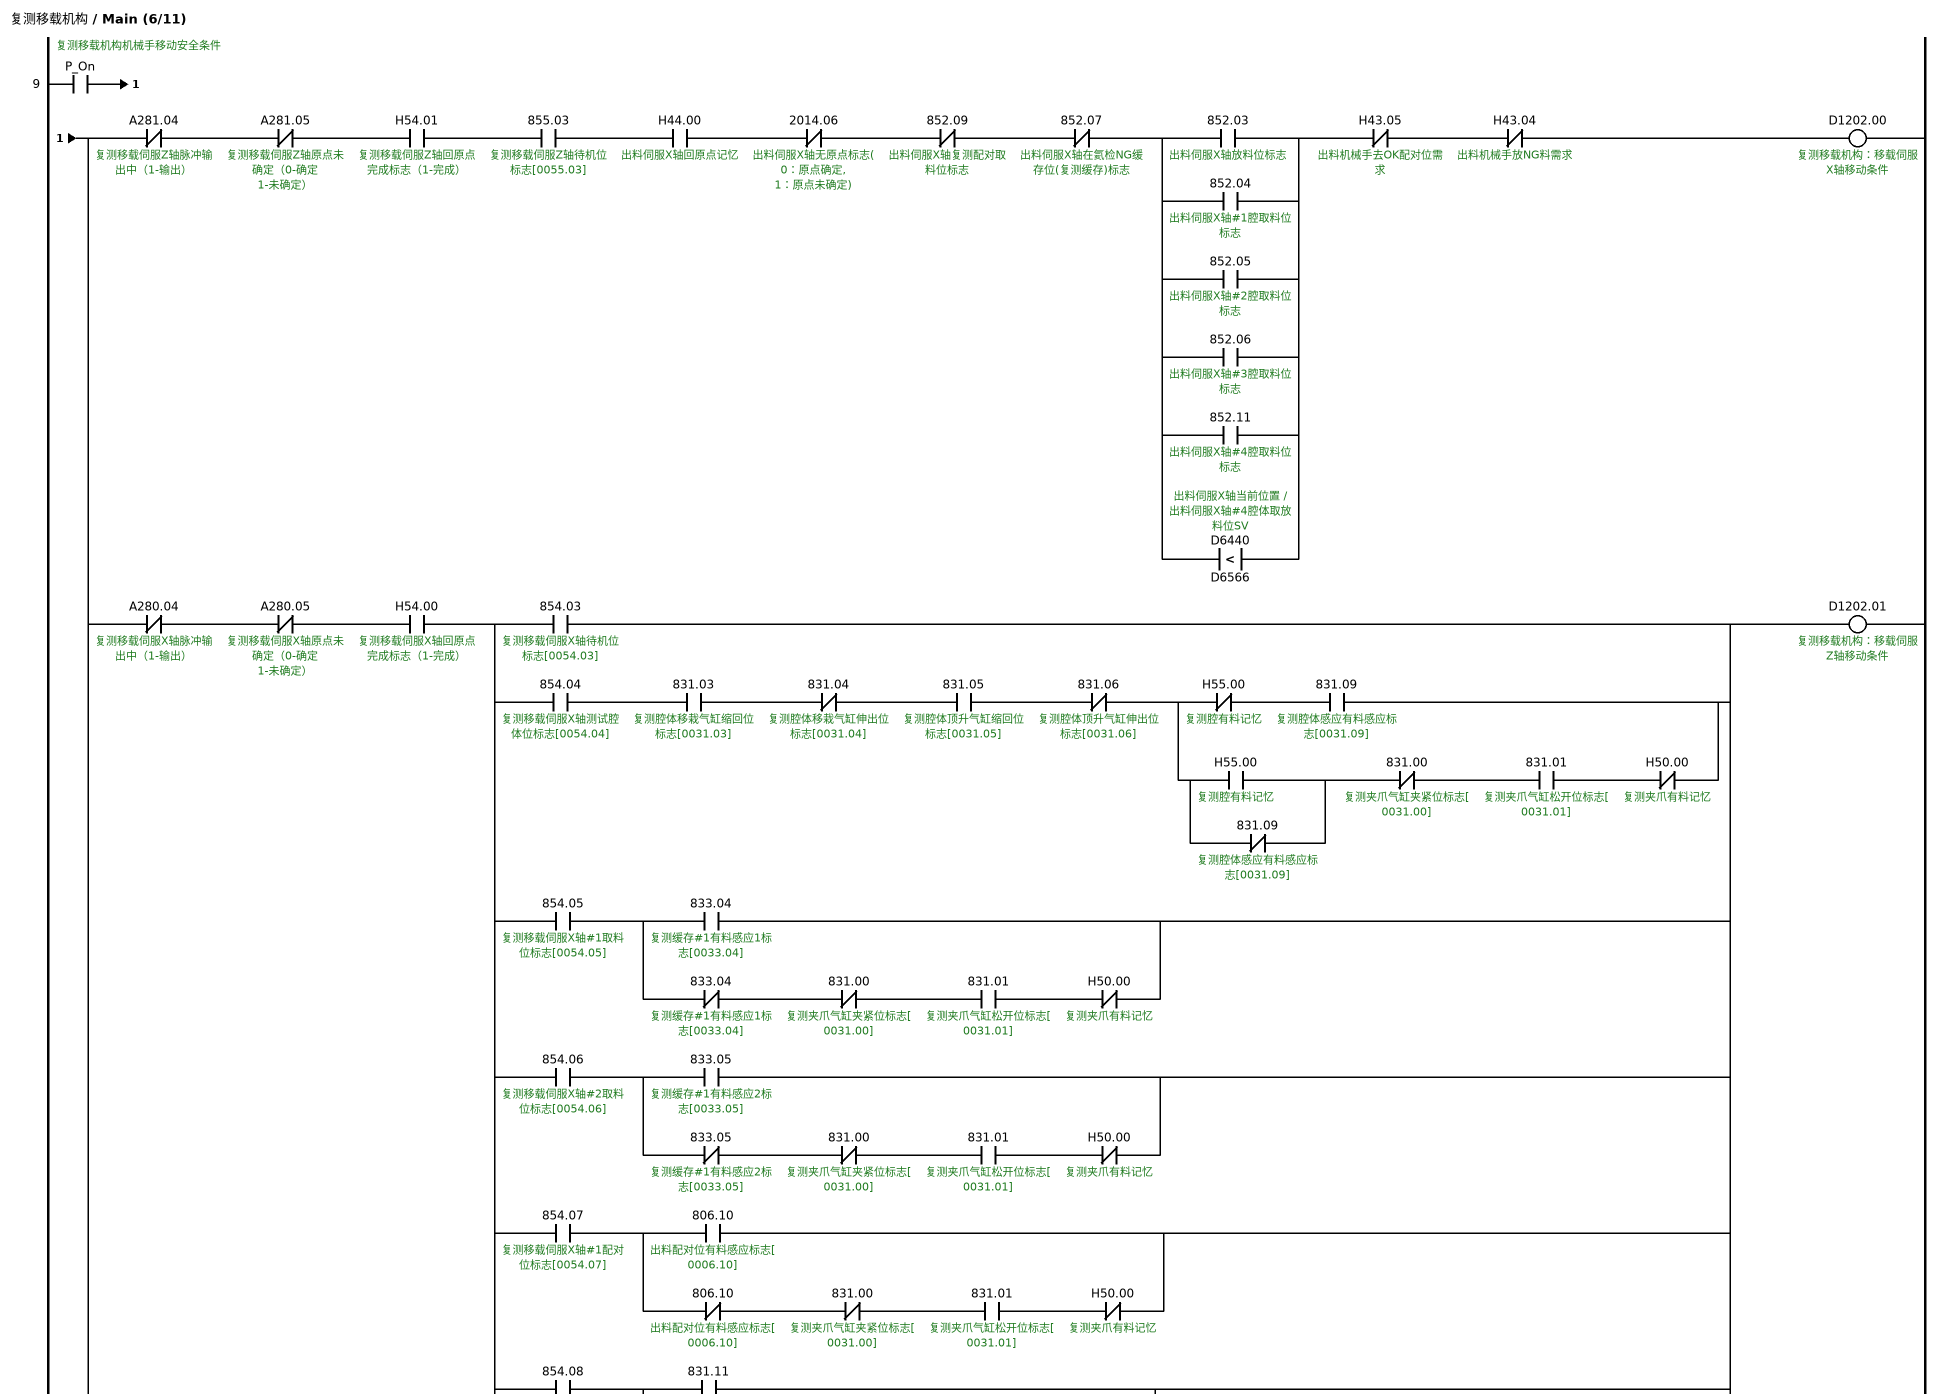

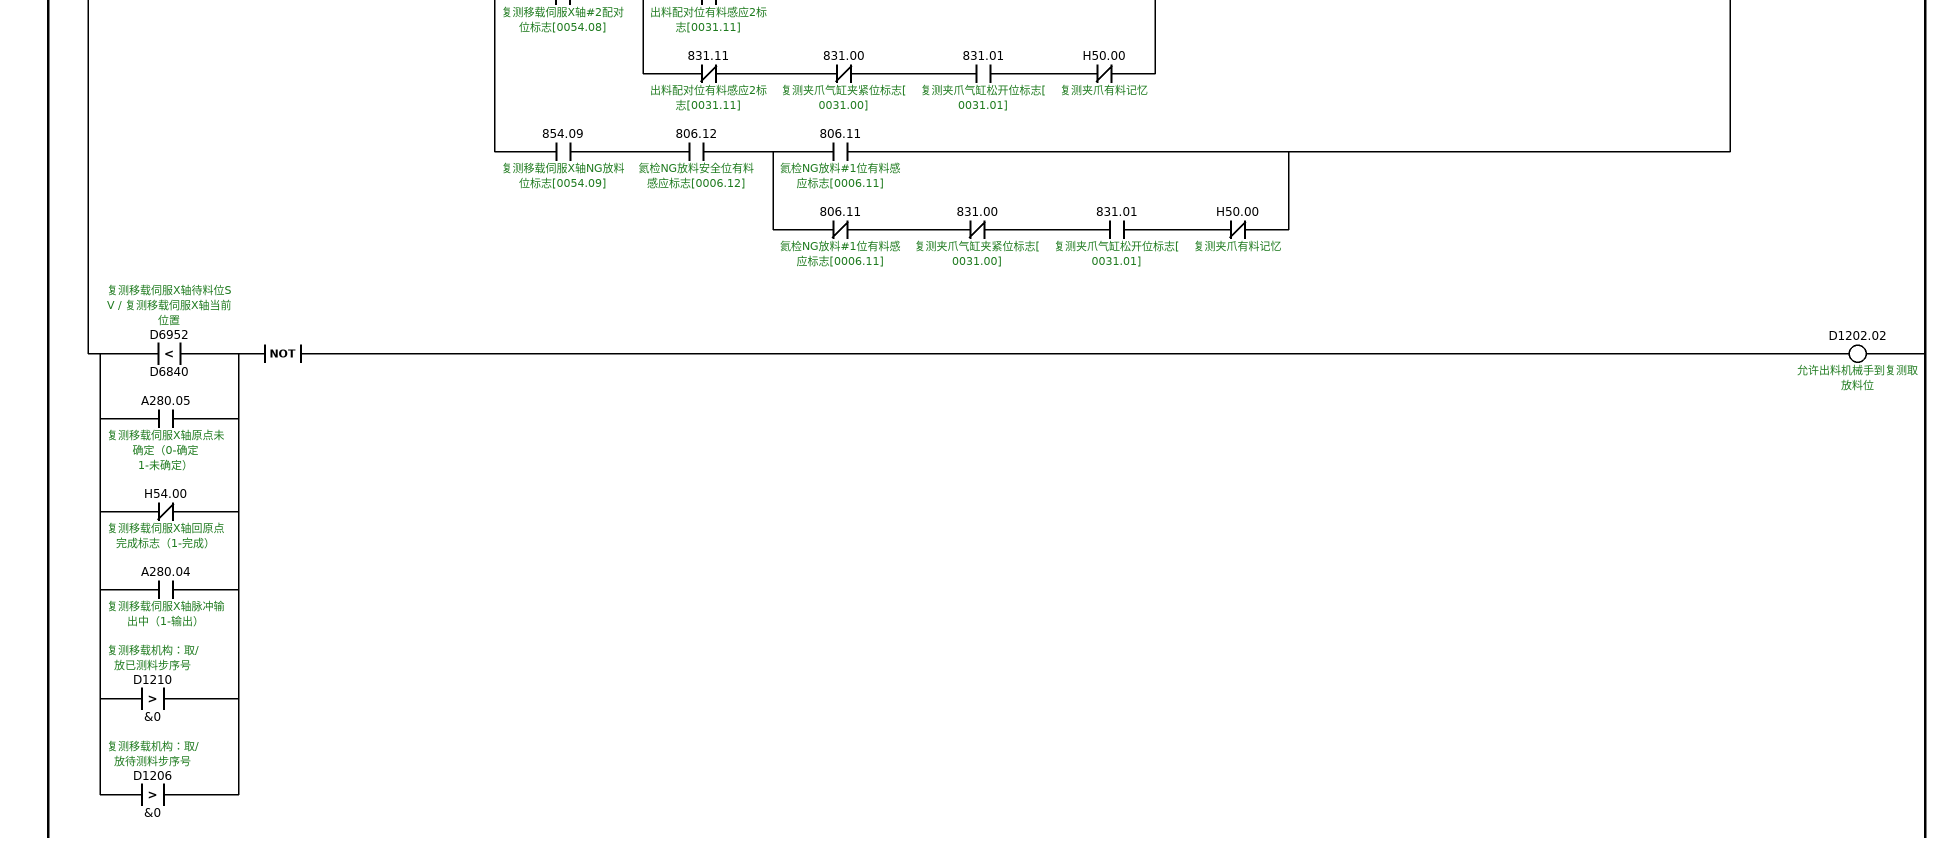
; rung 9: 复测移载机构机械手移动安全条件
LD P_On
OUT TR0
ANDNOT A281.04  ; 复测移载伺服Z轴脉冲输出中（1-输出）
ANDNOT A281.05  ; 复测移载伺服Z轴原点未确定（0-确定  1-未确定）
AND H54.01  ; 复测移载伺服Z轴回原点完成标志（1-完成）
AND 855.03  ; 复测移载伺服Z轴待机位标志[0055.03]
AND H44.00  ; 出料伺服X轴回原点记忆
ANDNOT 2014.06  ; 出料伺服X轴无原点标志(0：原点确定,1：原点未确定)
ANDNOT 852.09  ; 出料伺服X轴复测配对取料位标志
ANDNOT 852.07  ; 出料伺服X轴在氦检NG缓存位(复测缓存)标志
LD 852.03  ; 出料伺服X轴放料位标志
OR 852.04  ; 出料伺服X轴#1腔取料位标志
OR 852.05  ; 出料伺服X轴#2腔取料位标志
OR 852.06  ; 出料伺服X轴#3腔取料位标志
OR 852.11  ; 出料伺服X轴#4腔取料位标志
OR<SL(313) D6440 D6566  ; 出料伺服X轴当前位置, 出料伺服X轴#4腔体取放料位SV
ANDLD
ANDNOT H43.05  ; 出料机械手去OK配对位需求
ANDNOT H43.04  ; 出料机械手放NG料需求
OUT D1202.00  ; 复测移载机构：移载伺服X轴移动条件
LD TR0
ANDNOT A280.04  ; 复测移载伺服X轴脉冲输出中（1-输出）
ANDNOT A280.05  ; 复测移载伺服X轴原点未确定（0-确定  1-未确定）
AND H54.00  ; 复测移载伺服X轴回原点完成标志（1-完成）
LD 854.03  ; 复测移载伺服X轴待机位标志[0054.03]
LD 854.04  ; 复测移载伺服X轴测试腔体位标志[0054.04]
AND 831.03  ; 复测腔体移栽气缸缩回位标志[0031.03]
ANDNOT 831.04  ; 复测腔体移栽气缸伸出位标志[0031.04]
AND 831.05  ; 复测腔体顶升气缸缩回位标志[0031.05]
ANDNOT 831.06  ; 复测腔体顶升气缸伸出位标志[0031.06]
LDNOT H55.00  ; 复测腔有料记忆
AND 831.09  ; 复测腔体感应有料感应标志[0031.09]
LD H55.00  ; 复测腔有料记忆
ORNOT 831.09  ; 复测腔体感应有料感应标志[0031.09]
ANDNOT 831.00  ; 复测夹爪气缸夹紧位标志[0031.00]
AND 831.01  ; 复测夹爪气缸松开位标志[0031.01]
ANDNOT H50.00  ; 复测夹爪有料记忆
ORLD
ANDLD
ORLD
LD 854.05  ; 复测移载伺服X轴#1取料位标志[0054.05]
LD 833.04  ; 复测缓存#1有料感应1标志[0033.04]
LDNOT 833.04  ; 复测缓存#1有料感应1标志[0033.04]
ANDNOT 831.00  ; 复测夹爪气缸夹紧位标志[0031.00]
AND 831.01  ; 复测夹爪气缸松开位标志[0031.01]
ANDNOT H50.00  ; 复测夹爪有料记忆
ORLD
ANDLD
ORLD
LD 854.06  ; 复测移载伺服X轴#2取料位标志[0054.06]
LD 833.05  ; 复测缓存#1有料感应2标志[0033.05]
LDNOT 833.05  ; 复测缓存#1有料感应2标志[0033.05]
ANDNOT 831.00  ; 复测夹爪气缸夹紧位标志[0031.00]
AND 831.01  ; 复测夹爪气缸松开位标志[0031.01]
ANDNOT H50.00  ; 复测夹爪有料记忆
ORLD
ANDLD
ORLD
LD 854.07  ; 复测移载伺服X轴#1配对位标志[0054.07]
LD 806.10  ; 出料配对位有料感应标志[0006.10]
LDNOT 806.10  ; 出料配对位有料感应标志[0006.10]
ANDNOT 831.00  ; 复测夹爪气缸夹紧位标志[0031.00]
AND 831.01  ; 复测夹爪气缸松开位标志[0031.01]
ANDNOT H50.00  ; 复测夹爪有料记忆
ORLD
ANDLD
ORLD
LD 854.08  ; 复测移载伺服X轴#2配对位标志[0054.08]
LD 831.11  ; 出料配对位有料感应2标志[0031.11]
LDNOT 831.11  ; 出料配对位有料感应2标志[0031.11]
ANDNOT 831.00  ; 复测夹爪气缸夹紧位标志[0031.00]
AND 831.01  ; 复测夹爪气缸松开位标志[0031.01]
ANDNOT H50.00  ; 复测夹爪有料记忆
ORLD
ANDLD
ORLD
LD 854.09  ; 复测移载伺服X轴NG放料位标志[0054.09]
AND 806.12  ; 氦检NG放料安全位有料感应标志[0006.12]
LD 806.11  ; 氦检NG放料#1位有料感应标志[0006.11]
LDNOT 806.11  ; 氦检NG放料#1位有料感应标志[0006.11]
ANDNOT 831.00  ; 复测夹爪气缸夹紧位标志[0031.00]
AND 831.01  ; 复测夹爪气缸松开位标志[0031.01]
ANDNOT H50.00  ; 复测夹爪有料记忆
ORLD
ANDLD
ORLD
ANDLD
OUT D1202.01  ; 复测移载机构：移载伺服Z轴移动条件
LD TR0
LD<SL(313) D6952 D6840  ; 复测移载伺服X轴待料位SV, 复测移载伺服X轴当前位置
OR A280.05  ; 复测移载伺服X轴原点未确定（0-确定  1-未确定）
ORNOT H54.00  ; 复测移载伺服X轴回原点完成标志（1-完成）
OR A280.04  ; 复测移载伺服X轴脉冲输出中（1-输出）
OR>L(321) D1210 &0  ; 复测移载机构：取/放已测料步序号
OR>L(321) D1206 &0  ; 复测移载机构：取/放待测料步序号
ANDLD
NOT(520)
OUT D1202.02  ; 允许出料机械手到复测取放料位

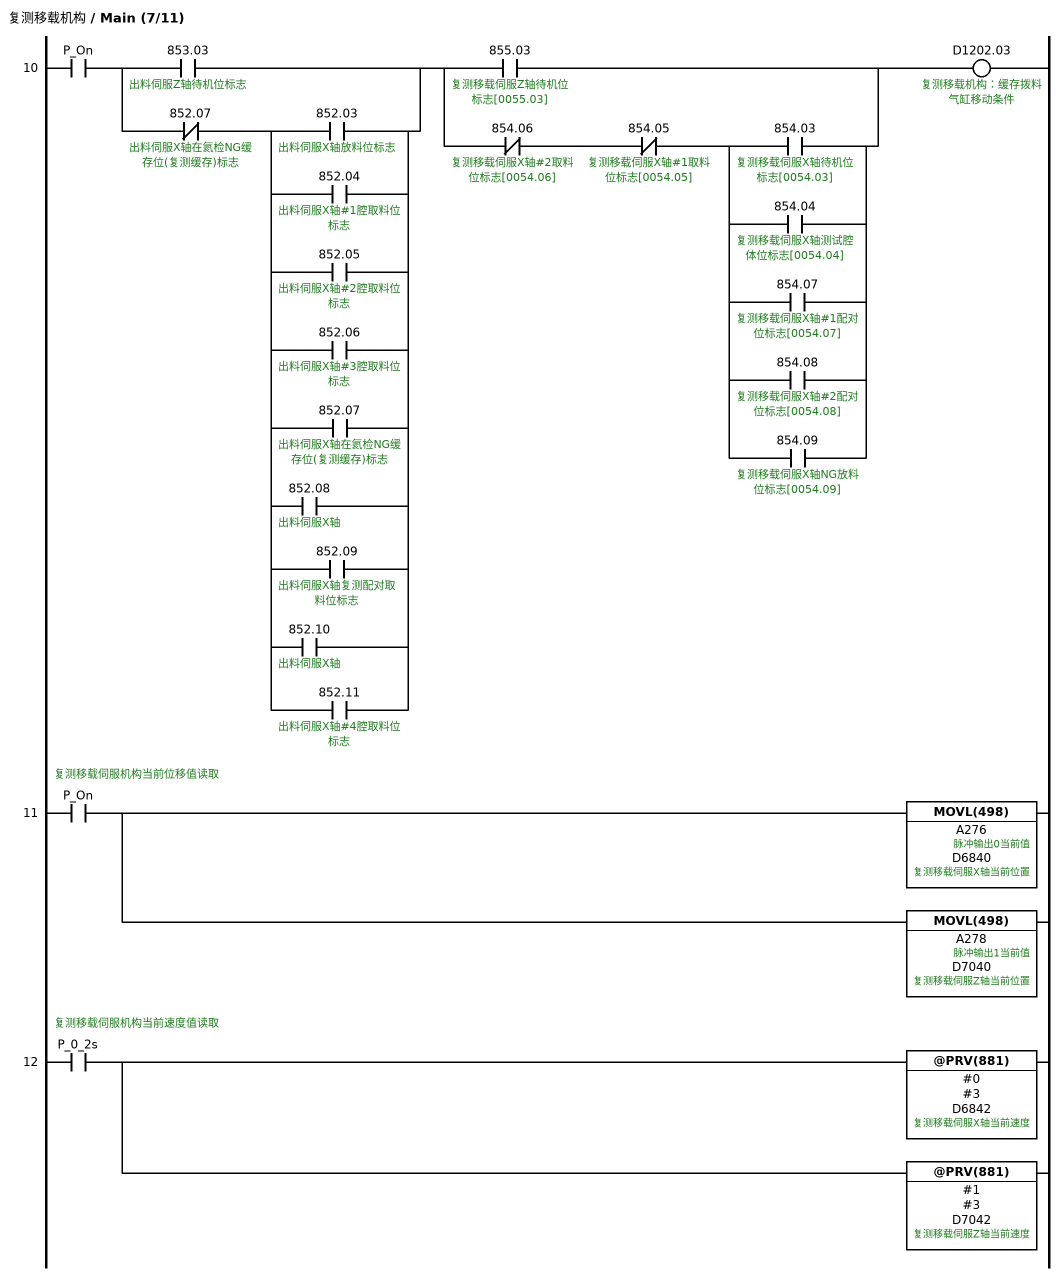
; rung 10
LD P_On
LD 853.03  ; 出料伺服Z轴待机位标志
LDNOT 852.07  ; 出料伺服X轴在氦检NG缓存位(复测缓存)标志  // 出料机械手不在缓存位
LD 852.03  ; 出料伺服X轴放料位标志
OR 852.04  ; 出料伺服X轴#1腔取料位标志
OR 852.05  ; 出料伺服X轴#2腔取料位标志
OR 852.06  ; 出料伺服X轴#3腔取料位标志
OR 852.07  ; 出料伺服X轴在氦检NG缓存位(复测缓存)标志
OR 852.08  ; 出料伺服X轴
OR 852.09  ; 出料伺服X轴复测配对取料位标志
OR 852.10  ; 出料伺服X轴
OR 852.11  ; 出料伺服X轴#4腔取料位标志
ANDLD
ORLD
ANDLD
LD 855.03  ; 复测移载伺服Z轴待机位标志[0055.03]
LDNOT 854.06  ; 复测移载伺服X轴#2取料位标志[0054.06]
ANDNOT 854.05  ; 复测移载伺服X轴#1取料位标志[0054.05]
LD 854.03  ; 复测移载伺服X轴待机位标志[0054.03]
OR 854.04  ; 复测移载伺服X轴测试腔体位标志[0054.04]
OR 854.07  ; 复测移载伺服X轴#1配对位标志[0054.07]
OR 854.08  ; 复测移载伺服X轴#2配对位标志[0054.08]
OR 854.09  ; 复测移载伺服X轴NG放料位标志[0054.09]
ANDLD
ORLD
ANDLD
OUT D1202.03  ; 复测移载机构：缓存拨料气缸移动条件
; rung 11: 复测移载伺服机构当前位移值读取
LD P_On
MOVL(498) A276 D6840  ; 脉冲输出0当前值, 复测移载伺服X轴当前位置
MOVL(498) A278 D7040  ; 脉冲输出1当前值, 复测移载伺服Z轴当前位置
; rung 12: 复测移载伺服机构当前速度值读取
LD P_0_2s
@PRV(881) #0 #3 D6842  ; 复测移载伺服X轴当前速度
@PRV(881) #1 #3 D7042  ; 复测移载伺服Z轴当前速度

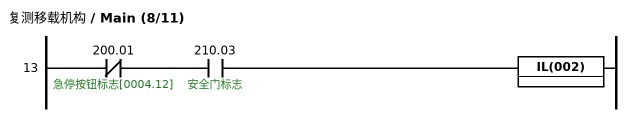
; rung 13
LDNOT 200.01  ; 急停按钮标志[0004.12]
AND 210.03  ; 安全门标志
IL(002)

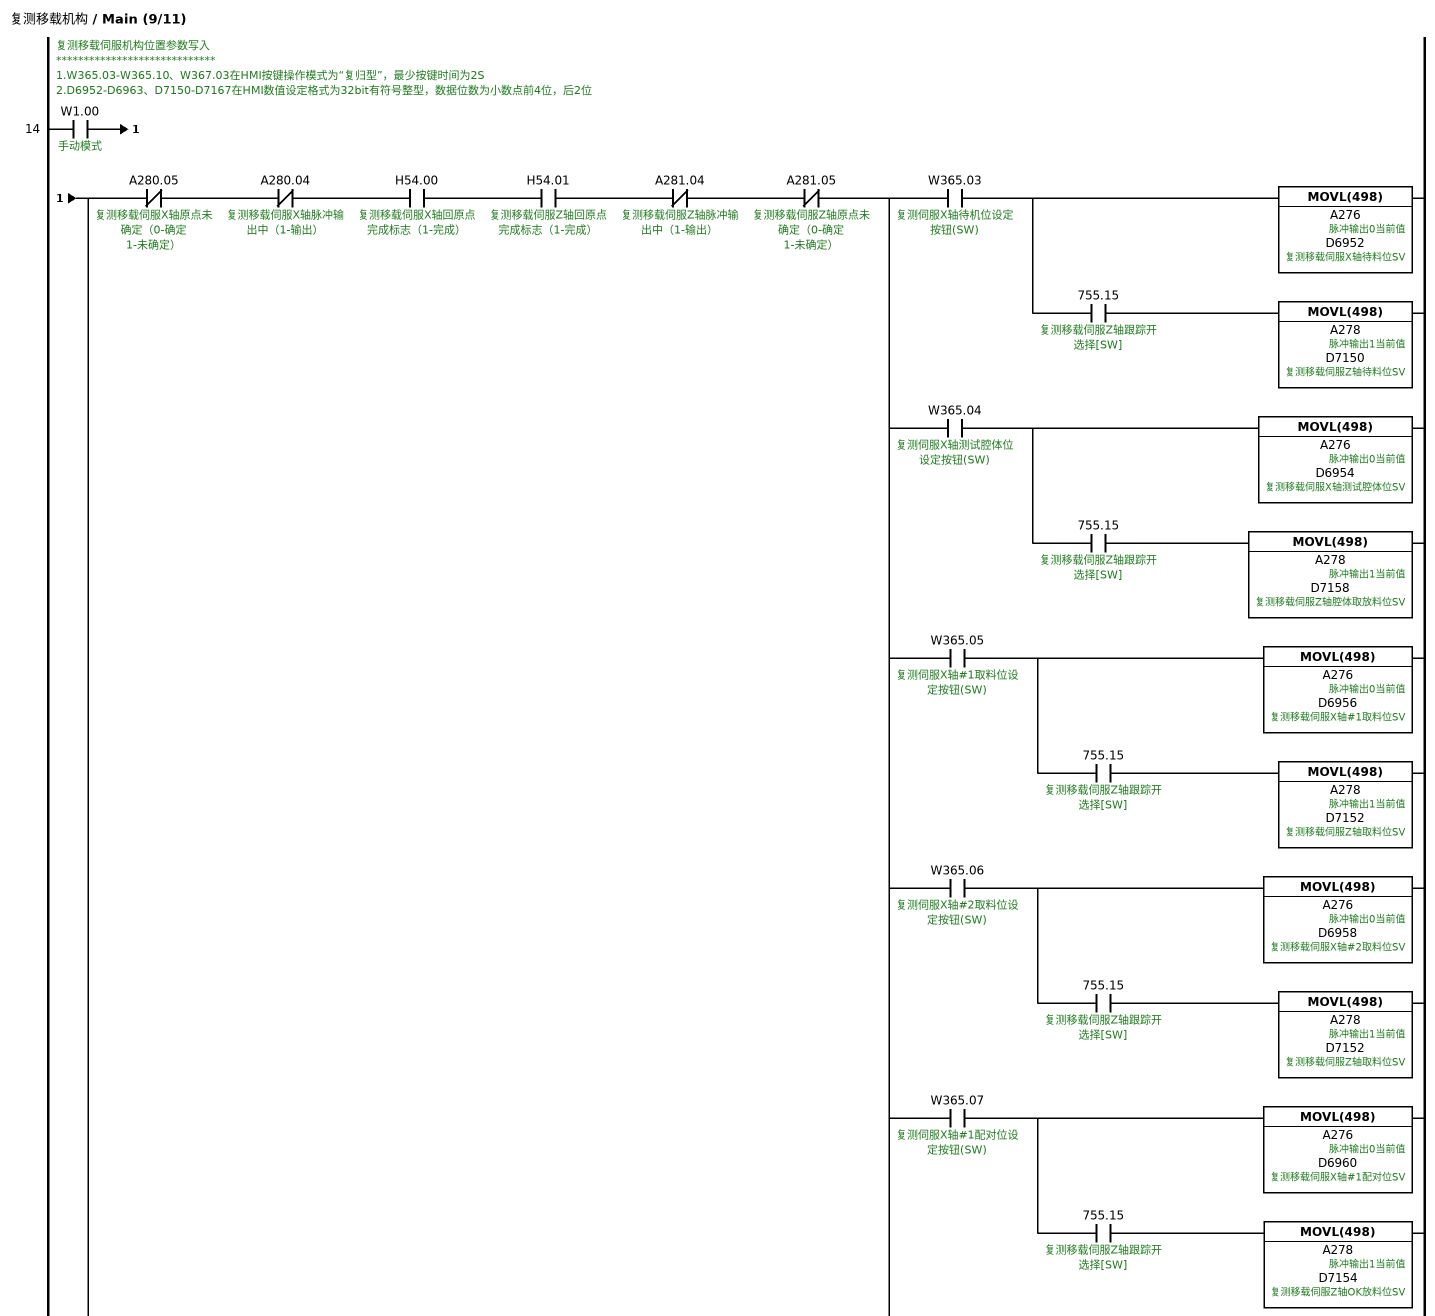

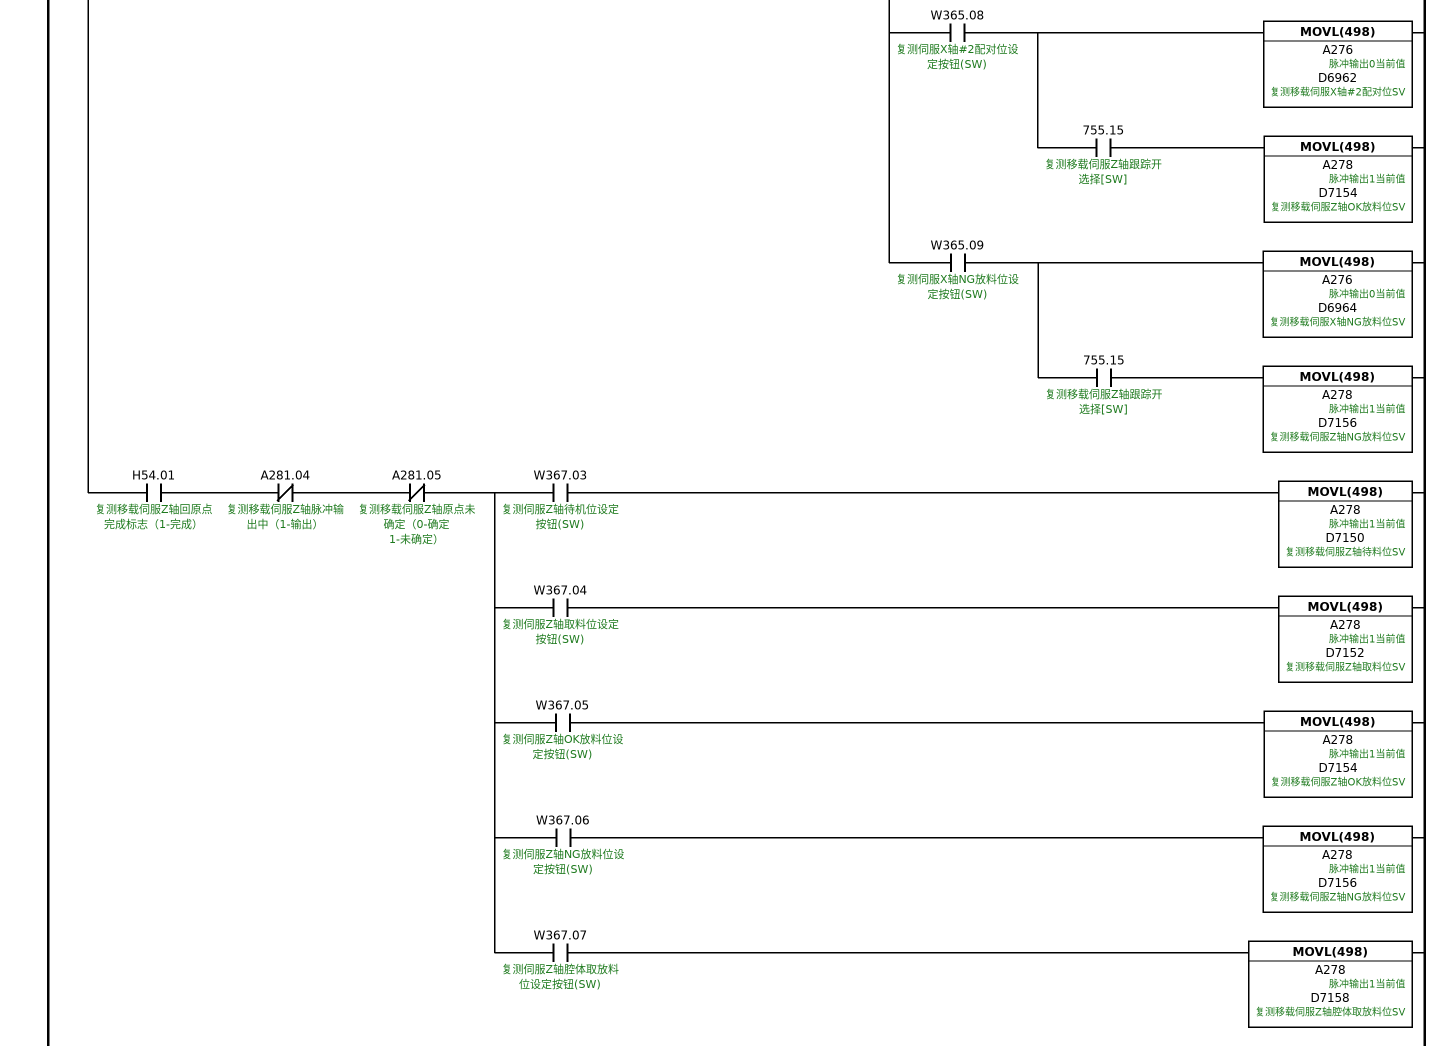
; rung 14: 复测移载伺服机构位置参数写入 / ***************************** / 1.W365.03-W365.10、W367.03在HMI按键操作模式为“复归型”，最少按键时间为2S / 2.D6952-D6963、D7150-D7167在HMI数值设定格式为32bit有符号整型，数据位数为小数点前4位，后2位
LD W1.00  ; 手动模式
OUT TR0
ANDNOT A280.05  ; 复测移载伺服X轴原点未确定（0-确定  1-未确定）
ANDNOT A280.04  ; 复测移载伺服X轴脉冲输出中（1-输出）
AND H54.00  ; 复测移载伺服X轴回原点完成标志（1-完成）
AND H54.01  ; 复测移载伺服Z轴回原点完成标志（1-完成）
ANDNOT A281.04  ; 复测移载伺服Z轴脉冲输出中（1-输出）
ANDNOT A281.05  ; 复测移载伺服Z轴原点未确定（0-确定  1-未确定）
OUT TR1
AND W365.03  ; 复测伺服X轴待机位设定按钮(SW)
MOVL(498) A276 D6952  ; 脉冲输出0当前值, 复测移载伺服X轴待料位SV
AND 755.15  ; 复测移载伺服Z轴跟踪开选择[SW]
MOVL(498) A278 D7150  ; 脉冲输出1当前值, 复测移载伺服Z轴待料位SV
LD TR1
AND W365.04  ; 复测伺服X轴测试腔体位设定按钮(SW)
MOVL(498) A276 D6954  ; 脉冲输出0当前值, 复测移载伺服X轴测试腔体位SV
AND 755.15  ; 复测移载伺服Z轴跟踪开选择[SW]
MOVL(498) A278 D7158  ; 脉冲输出1当前值, 复测移载伺服Z轴腔体取放料位SV
LD TR1
AND W365.05  ; 复测伺服X轴#1取料位设定按钮(SW)
MOVL(498) A276 D6956  ; 脉冲输出0当前值, 复测移载伺服X轴#1取料位SV
AND 755.15  ; 复测移载伺服Z轴跟踪开选择[SW]
MOVL(498) A278 D7152  ; 脉冲输出1当前值, 复测移载伺服Z轴取料位SV
LD TR1
AND W365.06  ; 复测伺服X轴#2取料位设定按钮(SW)
MOVL(498) A276 D6958  ; 脉冲输出0当前值, 复测移载伺服X轴#2取料位SV
AND 755.15  ; 复测移载伺服Z轴跟踪开选择[SW]
MOVL(498) A278 D7152  ; 脉冲输出1当前值, 复测移载伺服Z轴取料位SV
LD TR1
AND W365.07  ; 复测伺服X轴#1配对位设定按钮(SW)
MOVL(498) A276 D6960  ; 脉冲输出0当前值, 复测移载伺服X轴#1配对位SV
AND 755.15  ; 复测移载伺服Z轴跟踪开选择[SW]
MOVL(498) A278 D7154  ; 脉冲输出1当前值, 复测移载伺服Z轴OK放料位SV
LD TR1
AND W365.08  ; 复测伺服X轴#2配对位设定按钮(SW)
MOVL(498) A276 D6962  ; 脉冲输出0当前值, 复测移载伺服X轴#2配对位SV
AND 755.15  ; 复测移载伺服Z轴跟踪开选择[SW]
MOVL(498) A278 D7154  ; 脉冲输出1当前值, 复测移载伺服Z轴OK放料位SV
LD TR1
AND W365.09  ; 复测伺服X轴NG放料位设定按钮(SW)
MOVL(498) A276 D6964  ; 脉冲输出0当前值, 复测移载伺服X轴NG放料位SV
AND 755.15  ; 复测移载伺服Z轴跟踪开选择[SW]
MOVL(498) A278 D7156  ; 脉冲输出1当前值, 复测移载伺服Z轴NG放料位SV
LD TR0
AND H54.01  ; 复测移载伺服Z轴回原点完成标志（1-完成）
ANDNOT A281.04  ; 复测移载伺服Z轴脉冲输出中（1-输出）
ANDNOT A281.05  ; 复测移载伺服Z轴原点未确定（0-确定  1-未确定）
OUT TR0
AND W367.03  ; 复测伺服Z轴待机位设定按钮(SW)
MOVL(498) A278 D7150  ; 脉冲输出1当前值, 复测移载伺服Z轴待料位SV
LD TR0
AND W367.04  ; 复测伺服Z轴取料位设定按钮(SW)
MOVL(498) A278 D7152  ; 脉冲输出1当前值, 复测移载伺服Z轴取料位SV
LD TR0
AND W367.05  ; 复测伺服Z轴OK放料位设定按钮(SW)
MOVL(498) A278 D7154  ; 脉冲输出1当前值, 复测移载伺服Z轴OK放料位SV
LD TR0
AND W367.06  ; 复测伺服Z轴NG放料位设定按钮(SW)
MOVL(498) A278 D7156  ; 脉冲输出1当前值, 复测移载伺服Z轴NG放料位SV
LD TR0
AND W367.07  ; 复测伺服Z轴腔体取放料位设定按钮(SW)
MOVL(498) A278 D7158  ; 脉冲输出1当前值, 复测移载伺服Z轴腔体取放料位SV

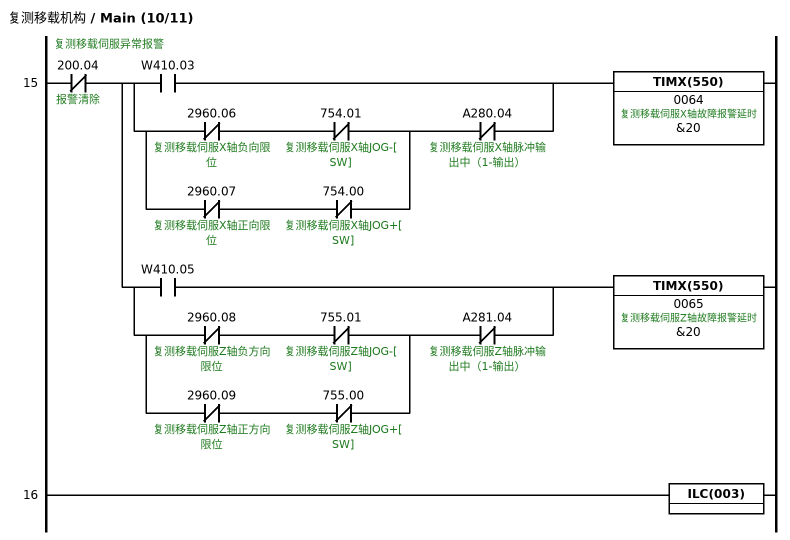
; rung 15: 复测移载伺服异常报警
LDNOT 200.04  ; 报警清除
OUT TR0
LD W410.03
LDNOT 2960.06  ; 复测移载伺服X轴负向限位
ANDNOT 754.01  ; 复测移载伺服X轴JOG-[SW]
LDNOT 2960.07  ; 复测移载伺服X轴正向限位
ANDNOT 754.00  ; 复测移载伺服X轴JOG+[SW]
ORLD
ANDNOT A280.04  ; 复测移载伺服X轴脉冲输出中（1-输出）
ORLD
ANDLD
TIMX(550) 0064 &20  ; 复测移载伺服X轴故障报警延时
LD TR0
LD W410.05
LDNOT 2960.08  ; 复测移载伺服Z轴负方向限位
ANDNOT 755.01  ; 复测移载伺服Z轴JOG-[SW]
LDNOT 2960.09  ; 复测移载伺服Z轴正方向限位
ANDNOT 755.00  ; 复测移载伺服Z轴JOG+[SW]
ORLD
ANDNOT A281.04  ; 复测移载伺服Z轴脉冲输出中（1-输出）
ORLD
ANDLD
TIMX(550) 0065 &20  ; 复测移载伺服Z轴故障报警延时
; rung 16
ILC(003)

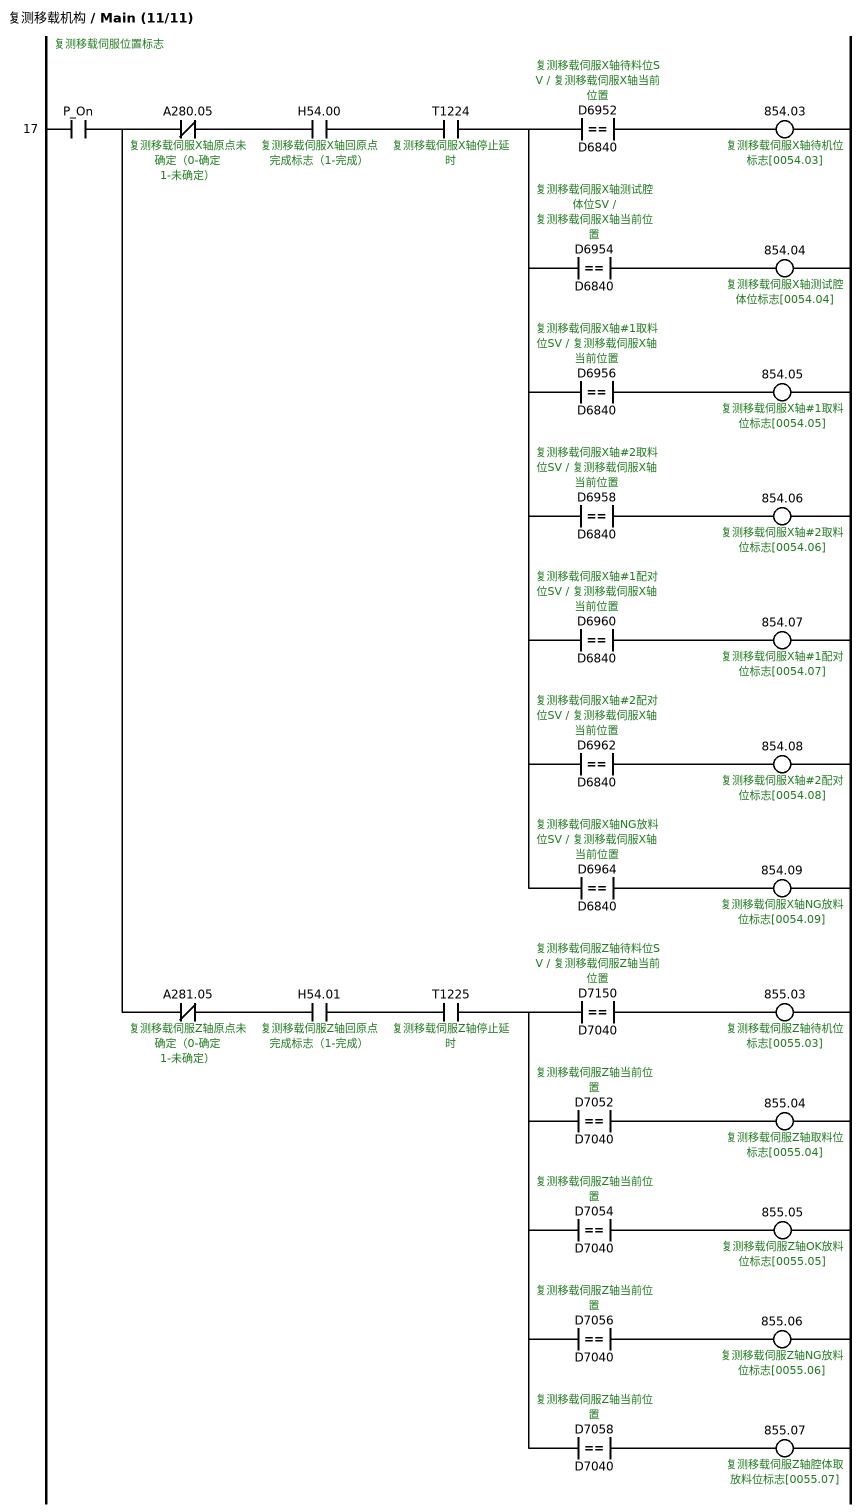
; rung 17: 复测移载伺服位置标志
LD P_On
OUT TR0
ANDNOT A280.05  ; 复测移载伺服X轴原点未确定（0-确定  1-未确定）
AND H54.00  ; 复测移载伺服X轴回原点完成标志（1-完成）
AND T1224  ; 复测移载伺服X轴停止延时
OUT TR1
AND=SL(303) D6952 D6840  ; 复测移载伺服X轴待料位SV, 复测移载伺服X轴当前位置
OUT 854.03  ; 复测移载伺服X轴待机位标志[0054.03]
LD TR1
AND=SL(303) D6954 D6840  ; 复测移载伺服X轴测试腔体位SV, 复测移载伺服X轴当前位置
OUT 854.04  ; 复测移载伺服X轴测试腔体位标志[0054.04]
LD TR1
AND=SL(303) D6956 D6840  ; 复测移载伺服X轴#1取料位SV, 复测移载伺服X轴当前位置
OUT 854.05  ; 复测移载伺服X轴#1取料位标志[0054.05]
LD TR1
AND=SL(303) D6958 D6840  ; 复测移载伺服X轴#2取料位SV, 复测移载伺服X轴当前位置
OUT 854.06  ; 复测移载伺服X轴#2取料位标志[0054.06]
LD TR1
AND=SL(303) D6960 D6840  ; 复测移载伺服X轴#1配对位SV, 复测移载伺服X轴当前位置
OUT 854.07  ; 复测移载伺服X轴#1配对位标志[0054.07]
LD TR1
AND=SL(303) D6962 D6840  ; 复测移载伺服X轴#2配对位SV, 复测移载伺服X轴当前位置
OUT 854.08  ; 复测移载伺服X轴#2配对位标志[0054.08]
LD TR1
AND=SL(303) D6964 D6840  ; 复测移载伺服X轴NG放料位SV, 复测移载伺服X轴当前位置
OUT 854.09  ; 复测移载伺服X轴NG放料位标志[0054.09]
LD TR0
ANDNOT A281.05  ; 复测移载伺服Z轴原点未确定（0-确定  1-未确定）
AND H54.01  ; 复测移载伺服Z轴回原点完成标志（1-完成）
AND T1225  ; 复测移载伺服Z轴停止延时
OUT TR0
AND=SL(303) D7150 D7040  ; 复测移载伺服Z轴待料位SV, 复测移载伺服Z轴当前位置
OUT 855.03  ; 复测移载伺服Z轴待机位标志[0055.03]
LD TR0
AND=SL(303) D7052 D7040  ; 复测移载伺服Z轴当前位置
OUT 855.04  ; 复测移载伺服Z轴取料位标志[0055.04]
LD TR0
AND=SL(303) D7054 D7040  ; 复测移载伺服Z轴当前位置
OUT 855.05  ; 复测移载伺服Z轴OK放料位标志[0055.05]
LD TR0
AND=SL(303) D7056 D7040  ; 复测移载伺服Z轴当前位置
OUT 855.06  ; 复测移载伺服Z轴NG放料位标志[0055.06]
LD TR0
AND=SL(303) D7058 D7040  ; 复测移载伺服Z轴当前位置
OUT 855.07  ; 复测移载伺服Z轴腔体取放料位标志[0055.07]

### Section 复测移载机构自动

